(* CoDeSys 2.3.9.28 project: JHV-kovolis.pro *)
(* Libraries: Ethernet.lib 2.12.10 13:48:32, mod_com.lib 2.12.10 13:48:32, ModbusEthernet_04.lib 2.12.10 13:48:36, Standard.lib 2.12.10 13:48:34, SYSLIBCALLBACK.LIB 2.12.10 13:48:32 *)

(* PLC configuration (modules and I/O channels)
IN1 AT %IX0.0 [BOOLOnX_I] Ch_1 Digital input
IN2 AT %IX0.1 [BOOLOnX_I] Ch_2 Digital input
IN3 AT %IX0.2 [BOOLOnX_I] Ch_3 Digital input
IN4 AT %IX0.3 [BOOLOnX_I] Ch_4 Digital input
IN5 AT %IX0.4 [BOOLOnX_I] Ch_5 Digital input
IN6 AT %IX0.5 [BOOLOnX_I] Ch_6 Digital input
IN7 AT %IX0.6 [BOOLOnX_I] Ch_7 Digital input
IN8 AT %IX0.7 [BOOLOnX_I] Ch_8 Digital input
IN9 AT %IX0.8 [BOOLOnX_I] Ch_1 Digital input
IN10 AT %IX0.9 [BOOLOnX_I] Ch_2 Digital input
IN11 AT %IX0.10 [BOOLOnX_I] Ch_3 Digital input
IN12 AT %IX0.11 [BOOLOnX_I] Ch_4 Digital input
IN13 AT %IX0.12 [BOOLOnX_I] Ch_5 Digital input
IN14 AT %IX0.13 [BOOLOnX_I] Ch_6 Digital input
IN15 AT %IX0.14 [BOOLOnX_I] Ch_7 Digital input
IN16 AT %IX0.15 [BOOLOnX_I] Ch_8 Digital input
Fieldbus variables [FB_VARS] node 1, in %IB0 out %QB0
*)

(* Global variable list: Global_Variables *)
VAR_GLOBAL
	IPHost1: STRING:= '192.168.0.100';
	IPHost2: STRING:= '192.168.0.101';

	Host1IN1: BOOL:= FALSE;
	Host1IN2: BOOL:= FALSE;
	Host1IN3: BOOL:= FALSE;
	Host1IN4: BOOL:= FALSE;
	Host1IN5: BOOL:= FALSE;
	Host1IN6: BOOL:= FALSE;
	Host1IN7: BOOL:= FALSE;
	Host1IN8: BOOL:= FALSE;

	Host2IN1: BOOL:= FALSE;
	Host2IN2: BOOL:= FALSE;
	Host2IN3: BOOL:= FALSE;
	Host2IN4: BOOL:= FALSE;
	Host2IN5: BOOL:= FALSE;
	Host2IN6: BOOL:= FALSE;
	Host2IN7: BOOL:= FALSE;
	Host2IN8: BOOL:= FALSE;

	OJS1: ARRAY [1..12] OF STRING;
	OJS2: ARRAY [1..8] OF STRING;
	OJS3: ARRAY [1..16] OF STRING;
	xOJS1: ARRAY [1..12] OF BOOL;
	xOJS2: ARRAY [1..8] OF BOOL;
	xOJS3: ARRAY [1..16] OF BOOL;
	xxOJS1: ARRAY [1..12] OF BOOL; (*Pøevrácená hodnota xOJS1*)
	xxOJS2: ARRAY [1..8] OF BOOL;	(*Pøevrácená hodnota xOJS2*)
	xxOJS3: ARRAY [1..16] OF BOOL;	(*Pøevrácená hodnota xOJS3*)

END_VAR

(* POU PLC_PRG, FBD *)
PROGRAM PLC_PRG
VAR
	Komunikace1: SlaveUDP_IO;
	Komunikace2: SlaveUDP_IO;
	sendStrHost1: ARRAY [1..100] OF WORD;
	sendStrHost2: ARRAY [1..100] OF WORD;
	RecStrHost1: ARRAY [1..100] OF WORD;
	RecStrHost2: ARRAY [1..100] OF WORD;
	Init1: BOOL;
	Init2: BOOL;
	NOERROR1: BOOL;
	NOERROR2: BOOL;
	PrevodnikHost1: WORD_TO_BOOL_16b;
	PrevodnikHost2: WORD_TO_BOOL_16b;
	Slitina: ARRAY [1..2] OF STRING:= 'Slitina1','Slitina2';
END_VAR
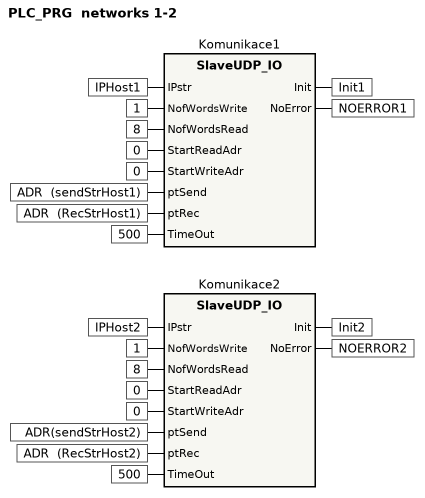
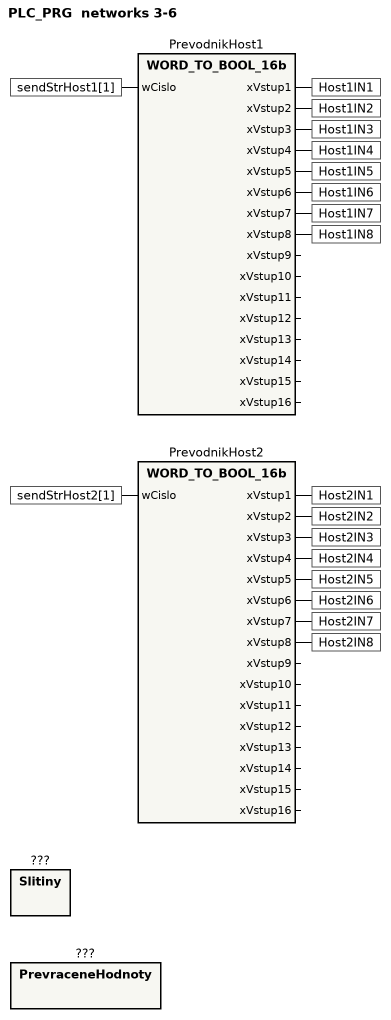
_FBD_ (* Function Block Diagram *)
NETWORK 1
	Komunikace1:SlaveUDP_IO(IPstr: IPHost1, NofWordsWrite: 1, NofWordsRead: 8, StartReadAdr: 0, StartWriteAdr: 0, ptSend: ADR	(sendStrHost1), ptRec: ADR	(RecStrHost1), TimeOut: 500, NoError => NOERROR1) => Init1
NETWORK 2
	Komunikace2:SlaveUDP_IO(IPstr: IPHost2, NofWordsWrite: 1, NofWordsRead: 8, StartReadAdr: 0, StartWriteAdr: 0, ptSend: 	ADR(sendStrHost2), ptRec: ADR	(RecStrHost2), TimeOut: 500, NoError => NOERROR2) => Init2
NETWORK 3
	PrevodnikHost1:WORD_TO_BOOL_16b(wCislo: sendStrHost1[1], xVstup2 => Host1IN2, xVstup3 => Host1IN3, xVstup4 => Host1IN4, xVstup5 => Host1IN5, xVstup6 => Host1IN6, xVstup7 => Host1IN7, xVstup8 => Host1IN8) => Host1IN1
NETWORK 4
	PrevodnikHost2:WORD_TO_BOOL_16b(wCislo: sendStrHost2[1], xVstup2 => Host2IN2, xVstup3 => Host2IN3, xVstup4 => Host2IN4, xVstup5 => Host2IN5, xVstup6 => Host2IN6, xVstup7 => Host2IN7, xVstup8 => Host2IN8) => Host2IN1
NETWORK 5
	???:Slitiny()
NETWORK 6
	???:PrevraceneHodnoty()
_END_FBD_
(* the same logic as Structured Text *)
(* Network 1 *)
Komunikace1(IPstr := IPHost1, NofWordsWrite := 1, NofWordsRead := 8, StartReadAdr := 0, StartWriteAdr := 0, ptSend := ADR	(sendStrHost1), ptRec := ADR	(RecStrHost1), TimeOut := 500);
NOERROR1 := Komunikace1.NoError;
Init1 := Komunikace1.Init;
(* Network 2 *)
Komunikace2(IPstr := IPHost2, NofWordsWrite := 1, NofWordsRead := 8, StartReadAdr := 0, StartWriteAdr := 0, ptSend := 	ADR(sendStrHost2), ptRec := ADR	(RecStrHost2), TimeOut := 500);
NOERROR2 := Komunikace2.NoError;
Init2 := Komunikace2.Init;
(* Network 3 *)
PrevodnikHost1(wCislo := sendStrHost1[1]);
Host1IN2 := PrevodnikHost1.xVstup2;
Host1IN3 := PrevodnikHost1.xVstup3;
Host1IN4 := PrevodnikHost1.xVstup4;
Host1IN5 := PrevodnikHost1.xVstup5;
Host1IN6 := PrevodnikHost1.xVstup6;
Host1IN7 := PrevodnikHost1.xVstup7;
Host1IN8 := PrevodnikHost1.xVstup8;
Host1IN1 := PrevodnikHost1.xVstup1;
(* Network 4 *)
PrevodnikHost2(wCislo := sendStrHost2[1]);
Host2IN2 := PrevodnikHost2.xVstup2;
Host2IN3 := PrevodnikHost2.xVstup3;
Host2IN4 := PrevodnikHost2.xVstup4;
Host2IN5 := PrevodnikHost2.xVstup5;
Host2IN6 := PrevodnikHost2.xVstup6;
Host2IN7 := PrevodnikHost2.xVstup7;
Host2IN8 := PrevodnikHost2.xVstup8;
Host2IN1 := PrevodnikHost2.xVstup1;
(* Network 5: see the listing above *)
(* Network 6: see the listing above *)
END_PROGRAM

(* POU SlaveUDP_IO, ST *)
FUNCTION_BLOCK SlaveUDP_IO
VAR_INPUT
	IPstr:STRING;					(*IP adresa slavu - 750-352,speedwaz etc.*)
	NofWordsWrite:WORD;		(*Pocet wordu, ktere maji byt zapsany*)
	NofWordsRead:WORD;		(*Pocet wordu, tkere maji byt cteny*)
	StartReadAdr:WORD;			(*adresa odkud se bude cist*)
	StartWriteAdr:WORD;			(*odresa kam se bude zapisovat*)
	ptSend:POINTER TO WORD;	(*pointer na pole ktere se bude zapisovat*)
	ptRec:POINTER TO WORD;	(*pointer na pole ktere se bude cist*)
	TimeOut:WORD:=500;		(*cas v milisekundach, pokud neni zadna komunikace, tak potomto case se vystupy nastavi do nuly*)
END_VAR
VAR_OUTPUT
	Init:BOOL;					(*cas do watchdogu byl zapsan a watchdog je spusten -> je mozne komunikovat*)
	NoError:BOOL;			(*zadna chyba pri komunikaci*)
END_VAR
VAR
	state:INT:=0;
	master882: ETHERNET_MODBUSMASTER_UDP;
	start882:BOOL:=FALSE;
	res882:BOOL:=FALSE;
	err882:WORD;
	ready882:BOOL;
	resp882:BYTE;
	ftrig882: F_TRIG;
	tmp_val:WORD;

	ptWrite:POINTER TO BYTE;
	NofWrite:INT;
	WriteAdr:WORD;
END_VAR
IF start882=FALSE THEN
	start882:=TRUE;
	CASE state OF
		0:
			(*zastaveni casovace*)
			tmp_val:=0;
			WriteAdr:=16#100A;
			ptWrite:=ADR(tmp_val);
			NofWrite:=1;
		1:
			(*nastaveni casu, cas je mozne nastavit jen tehdy, kdyz je casovac zastaven*)
			TimeOut:=TimeOut/100;
			tmp_val:=TimeOut;
			NofWordsWrite:=1;
			WriteAdr:=16#1000;
			ptWrite:=ADR(tmp_val);
			NofWrite:=1;
		2:
			(*spusteni watchdogu*)
			tmp_val:=1;
			WriteAdr:=16#100A;
			ptWrite:=ADR(tmp_val);
			NofWrite:=1;
		3:
			(*bezna komunikace*)
			ptWrite:=ptSend;
			NofWrite:=NofWordsWrite;
			WriteAdr:=StartWriteAdr;
	END_CASE;
END_IF;

NofWordsRead;
NofWrite;
IF NofWrite=0 THEN
(*cteni 352 kdyz neni treba nic zapsat*)
master882(strIP_ADDRESS := IPstr,	wPORT := 502,bUNIT_ID := 0,bFUNCTION_CODE := 3,wREAD_ADDRESS := StartReadAdr,wREAD_QUANTITY :=NofWordsRead,
	ptREAD_DATA :=ptRec,wWRITE_ADDRESS := WriteAdr,wWRITE_QUANTITY := NofWrite,ptSEND_DATA :=ptWrite ,xSTART := start882,xRESET := res882,
	tTIME_OUT := t#1s);
ELSE
(*blok pro cteni i zapis v jednom cyklu*)
master882(strIP_ADDRESS := IPstr,	wPORT := 502,bUNIT_ID := 0,bFUNCTION_CODE := 23,wREAD_ADDRESS := StartReadAdr,wREAD_QUANTITY :=NofWordsRead,
	ptREAD_DATA :=ptRec,wWRITE_ADDRESS := WriteAdr,wWRITE_QUANTITY := NofWrite,ptSEND_DATA :=ptWrite ,xSTART := start882,xRESET := res882,
	tTIME_OUT := t#1s);
END_IF;
	(* vystupni promenne *)
	err882:=master882.wERROR;
	ready882:= master882.xREADY;
	resp882:=master882.bRESPONSE_UNIT_ID;

IF master882.wERROR=0 THEN
	NoError:=TRUE;
ELSE
	NoError:=FALSE;
END_IF;
ftrig882(clk:=ready882);
(*prechody ve stavovem automau*)
IF ftrig882.Q   THEN
	 start882:=FALSE;
	IF master882.wERROR=0 THEN
		state:=state+1;	(*neni chyba komunikace, prejdi do dalsiho stavu*)
	ELSE
		IF state>0 AND state<3 THEN
			(*nastala nejaka chyba, vrat so inicializace casovace*)
			state:=0;
		END_IF;
	END_IF;
	IF state>=3 THEN
		state:=3;
		init:=TRUE;
	END_IF;
END_IF;
END_FUNCTION_BLOCK

(* POU Komunikace/WORD_TO_BOOL_16b, ST *)
FUNCTION_BLOCK WORD_TO_BOOL_16b
VAR_INPUT
	wCislo: WORD;

END_VAR
VAR_OUTPUT
	xVstup1: BOOL;
	xVstup2: BOOL;
	xVstup3: BOOL;
	xVstup4: BOOL;
	xVstup5: BOOL;
	xVstup6: BOOL;
	xVstup7: BOOL;
	xVstup8: BOOL;
	xVstup9: BOOL;
	xVstup10: BOOL;
	xVstup11: BOOL;
	xVstup12: BOOL;
	xVstup13: BOOL;
	xVstup14: BOOL;
	xVstup15: BOOL;
	xVstup16: BOOL;
END_VAR
VAR
END_VAR
IF (wCislo > 0)
	THEN
		(*15tı bit*)
		IF(wCislo/32768 > 0)
			THEN
				xVstup16 := TRUE;
				wCislo:= wCislo - 32768;
		ELSE
				xVstup16 := FALSE;
		END_IF

		(*14tı bit*)
		IF(wCislo/16384 > 0)
			THEN
				xVstup15 := TRUE;
				wCislo:= wCislo - 16384;
		ELSE
				xVstup15 := FALSE;
		END_IF

		(*13tı bit*)
		IF(wCislo/8192 > 0)
			THEN
				xVstup14 := TRUE;
				wCislo:= wCislo - 8192;
		ELSE
				xVstup14 := FALSE;
		END_IF

		(*12tı bit*)
		IF(wCislo/4096 > 0)
			THEN
				xVstup13 := TRUE;
				wCislo:= wCislo - 4096;
		ELSE
				xVstup13 := FALSE;
		END_IF

		(*11tı bit*)
		IF(wCislo/2048 > 0)
			THEN
				xVstup12 := TRUE;
				wCislo:= wCislo - 2048;
		ELSE
				xVstup12 := FALSE;
		END_IF

		(*10tı bit*)
		IF(wCislo/1024 > 0)
			THEN
				xVstup11 := TRUE;
				wCislo:= wCislo - 1024;
		ELSE
				xVstup11 := FALSE;
		END_IF

		(*9tı bit*)
		IF(wCislo/512 > 0)
			THEN
				xVstup10 := TRUE;
				wCislo:= wCislo - 512;
		ELSE
				xVstup10 := FALSE;
		END_IF

		(*8tı bit*)
		IF(wCislo/256 > 0)
			THEN
				xVstup9 := TRUE;
				wCislo:= wCislo - 256;
		ELSE
				xVstup9 := FALSE;
		END_IF

		(*7tı bit*)
		IF(wCislo/128 > 0)
			THEN
				xVstup8 := TRUE;
				wCislo:= wCislo - 128;
		ELSE
				xVstup8 := FALSE;
		END_IF

		(*6tı bit*)
		IF(wCislo/64 > 0)
			THEN
				xVstup7 := TRUE;
				wCislo:= wCislo - 64;
		ELSE
				xVstup7 := FALSE;
		END_IF

		(*5tı bit*)
		IF(wCislo/32 > 0)
			THEN
				xVstup6 := TRUE;
				wCislo:= wCislo - 32;
		ELSE
				xVstup6 := FALSE;
		END_IF

		(*4tı bit*)
		IF(wCislo/16 > 0)
			THEN
				xVstup5 := TRUE;
				wCislo:= wCislo - 16;
		ELSE
				xVstup5 := FALSE;
		END_IF

		(*3tí bit*)
		IF(wCislo/8 > 0)
			THEN
				xVstup4 := TRUE;
				wCislo:= wCislo - 8;
		ELSE
				xVstup4 := FALSE;
		END_IF

		(*2hı bit*)
		IF(wCislo/4 > 0)
			THEN
				xVstup3 := TRUE;
				wCislo:= wCislo - 4;
		ELSE
				xVstup3 := FALSE;
		END_IF

		(*1ní bit*)
		IF(wCislo/2 > 0)
			THEN
				xVstup2 := TRUE;
				wCislo:= wCislo - 2;
		ELSE
				xVstup2 := FALSE;
		END_IF

		(*0tı bit*)
		IF(wCislo > 0)
			THEN
				xVstup1 := TRUE;
				wCislo:= wCislo - 1;
		ELSE
				xVstup1 := FALSE;
		END_IF
END_IF
END_FUNCTION_BLOCK

(* POU Slitiny/Slitiny, CFC *)
PROGRAM Slitiny
VAR
	s1: VybranaSlitina;
	s2: VybranaSlitina;
	s3: VybranaSlitina;
	s4: VybranaSlitina;
	s5: VybranaSlitina;
	s6: VybranaSlitina;
	s7: VybranaSlitina;
	s8: VybranaSlitina;
	s9: VybranaSlitina;
	s10: VybranaSlitina;
	s11: VybranaSlitina;
	s12: VybranaSlitina;

	s13: VybranaSlitina;
	s14: VybranaSlitina;
	s15: VybranaSlitina;
	s16: VybranaSlitina;
	s17: VybranaSlitina;
	s18: VybranaSlitina;
	s19: VybranaSlitina;
	s20: VybranaSlitina;

	s21: VybranaSlitina;
	s22: VybranaSlitina;
	s23: VybranaSlitina;
	s24: VybranaSlitina;
	s25: VybranaSlitina;
	s26: VybranaSlitina;
	s27: VybranaSlitina;
	s28: VybranaSlitina;
	s29: VybranaSlitina;
	s30: VybranaSlitina;
	s31: VybranaSlitina;
	s32: VybranaSlitina;
	s33: VybranaSlitina;
	s34: VybranaSlitina;
	s35: VybranaSlitina;
END_VAR
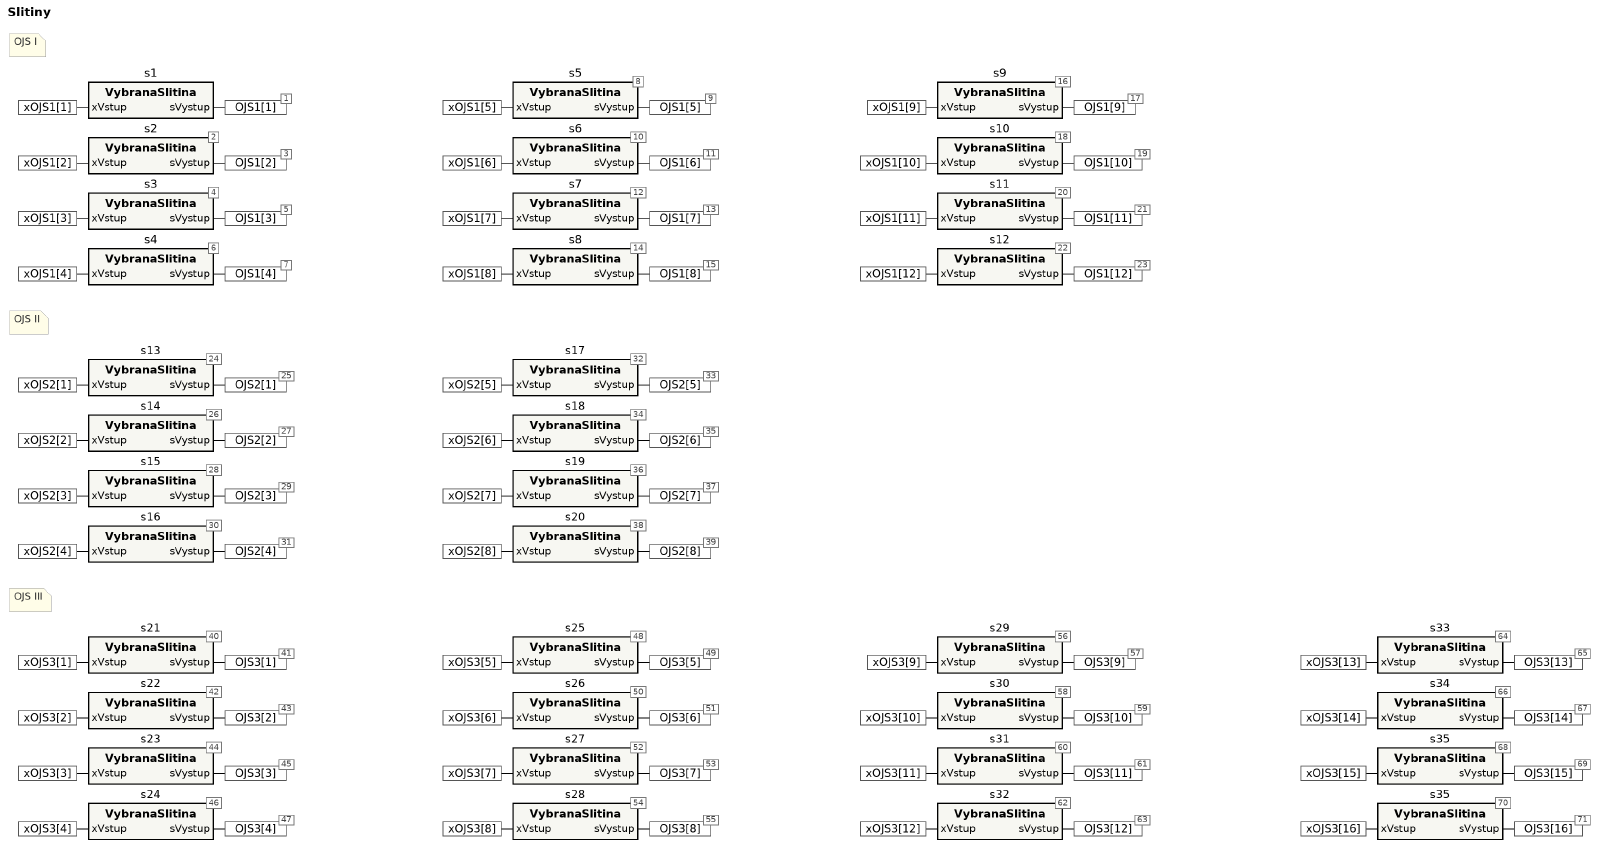
_CFC_ (* Continuous Function Chart, elements in execution order *)
(* OJS I *)
#0 s1:VybranaSlitina(xVstup: xOJS1[1])
#1 OJS1[1] <= #0.sVystup
#2 s2:VybranaSlitina(xVstup: xOJS1[2])
#3 OJS1[2] <= #2.sVystup
#4 s3:VybranaSlitina(xVstup: xOJS1[3])
#5 OJS1[3] <= #4.sVystup
#6 s4:VybranaSlitina(xVstup: xOJS1[4])
#7 OJS1[4] <= #6.sVystup
#8 s5:VybranaSlitina(xVstup: xOJS1[5])
#9 OJS1[5] <= #8.sVystup
#10 s6:VybranaSlitina(xVstup: xOJS1[6])
#11 OJS1[6] <= #10.sVystup
#12 s7:VybranaSlitina(xVstup: xOJS1[7])
#13 OJS1[7] <= #12.sVystup
#14 s8:VybranaSlitina(xVstup: xOJS1[8])
#15 OJS1[8] <= #14.sVystup
#16 s9:VybranaSlitina(xVstup: xOJS1[9])
#17 OJS1[9] <= #16.sVystup
#18 s10:VybranaSlitina(xVstup: xOJS1[10])
#19 OJS1[10] <= #18.sVystup
#20 s11:VybranaSlitina(xVstup: xOJS1[11])
#21 OJS1[11] <= #20.sVystup
#22 s12:VybranaSlitina(xVstup: xOJS1[12])
#23 OJS1[12] <= #22.sVystup
(* OJS II *)
#24 s13:VybranaSlitina(xVstup: xOJS2[1])
#25 OJS2[1] <= #24.sVystup
#26 s14:VybranaSlitina(xVstup: xOJS2[2])
#27 OJS2[2] <= #26.sVystup
#28 s15:VybranaSlitina(xVstup: xOJS2[3])
#29 OJS2[3] <= #28.sVystup
#30 s16:VybranaSlitina(xVstup: xOJS2[4])
#31 OJS2[4] <= #30.sVystup
#32 s17:VybranaSlitina(xVstup: xOJS2[5])
#33 OJS2[5] <= #32.sVystup
#34 s18:VybranaSlitina(xVstup: xOJS2[6])
#35 OJS2[6] <= #34.sVystup
#36 s19:VybranaSlitina(xVstup: xOJS2[7])
#37 OJS2[7] <= #36.sVystup
#38 s20:VybranaSlitina(xVstup: xOJS2[8])
#39 OJS2[8] <= #38.sVystup
(* OJS III *)
#40 s21:VybranaSlitina(xVstup: xOJS3[1])
#41 OJS3[1] <= #40.sVystup
#42 s22:VybranaSlitina(xVstup: xOJS3[2])
#43 OJS3[2] <= #42.sVystup
#44 s23:VybranaSlitina(xVstup: xOJS3[3])
#45 OJS3[3] <= #44.sVystup
#46 s24:VybranaSlitina(xVstup: xOJS3[4])
#47 OJS3[4] <= #46.sVystup
#48 s25:VybranaSlitina(xVstup: xOJS3[5])
#49 OJS3[5] <= #48.sVystup
#50 s26:VybranaSlitina(xVstup: xOJS3[6])
#51 OJS3[6] <= #50.sVystup
#52 s27:VybranaSlitina(xVstup: xOJS3[7])
#53 OJS3[7] <= #52.sVystup
#54 s28:VybranaSlitina(xVstup: xOJS3[8])
#55 OJS3[8] <= #54.sVystup
#56 s29:VybranaSlitina(xVstup: xOJS3[9])
#57 OJS3[9] <= #56.sVystup
#58 s30:VybranaSlitina(xVstup: xOJS3[10])
#59 OJS3[10] <= #58.sVystup
#60 s31:VybranaSlitina(xVstup: xOJS3[11])
#61 OJS3[11] <= #60.sVystup
#62 s32:VybranaSlitina(xVstup: xOJS3[12])
#63 OJS3[12] <= #62.sVystup
#64 s33:VybranaSlitina(xVstup: xOJS3[13])
#65 OJS3[13] <= #64.sVystup
#66 s34:VybranaSlitina(xVstup: xOJS3[14])
#67 OJS3[14] <= #66.sVystup
#68 s35:VybranaSlitina(xVstup: xOJS3[15])
#69 OJS3[15] <= #68.sVystup
#70 s35:VybranaSlitina(xVstup: xOJS3[16])
#71 OJS3[16] <= #70.sVystup
_END_CFC_
END_PROGRAM

(* POU Slitiny/VybranaSlitina, ST *)
FUNCTION_BLOCK VybranaSlitina
VAR_INPUT
	xVstup: BOOL;
END_VAR
VAR_OUTPUT
	sVystup: STRING;
END_VAR
VAR
END_VAR
IF (xVstup)
THEN
	sVystup:= PLC_PRG.Slitina[1];
ELSE
	sVystup:= PLC_PRG.Slitina[2];
END_IF
END_FUNCTION_BLOCK

(* POU Slitiny/PrevraceneHodnoty, CFC *)
PROGRAM PrevraceneHodnoty
VAR
END_VAR
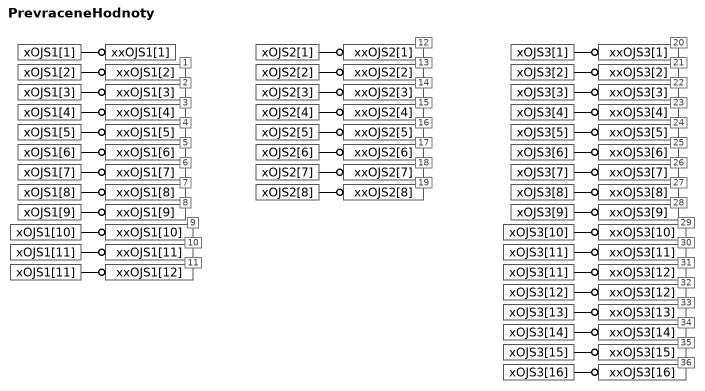
_CFC_ (* Continuous Function Chart, elements in execution order *)
#0 xxOJS1[1] <= NOT xOJS1[1]
#1 xxOJS1[2] <= NOT xOJS1[2]
#2 xxOJS1[3] <= NOT xOJS1[3]
#3 xxOJS1[4] <= NOT xOJS1[4]
#4 xxOJS1[5] <= NOT xOJS1[5]
#5 xxOJS1[6] <= NOT xOJS1[6]
#6 xxOJS1[7] <= NOT xOJS1[7]
#7 xxOJS1[8] <= NOT xOJS1[8]
#8 xxOJS1[9] <= NOT xOJS1[9]
#9 xxOJS1[10] <= NOT xOJS1[10]
#10 xxOJS1[11] <= NOT xOJS1[11]
#11 xxOJS1[12] <= NOT xOJS1[11]
#12 xxOJS2[1] <= NOT xOJS2[1]
#13 xxOJS2[2] <= NOT xOJS2[2]
#14 xxOJS2[3] <= NOT xOJS2[3]
#15 xxOJS2[4] <= NOT xOJS2[4]
#16 xxOJS2[5] <= NOT xOJS2[5]
#17 xxOJS2[6] <= NOT xOJS2[6]
#18 xxOJS2[7] <= NOT xOJS2[7]
#19 xxOJS2[8] <= NOT xOJS2[8]
#20 xxOJS3[1] <= NOT xOJS3[1]
#21 xxOJS3[2] <= NOT xOJS3[2]
#22 xxOJS3[3] <= NOT xOJS3[3]
#23 xxOJS3[4] <= NOT xOJS3[4]
#24 xxOJS3[5] <= NOT xOJS3[5]
#25 xxOJS3[6] <= NOT xOJS3[6]
#26 xxOJS3[7] <= NOT xOJS3[7]
#27 xxOJS3[8] <= NOT xOJS3[8]
#28 xxOJS3[9] <= NOT xOJS3[9]
#29 xxOJS3[10] <= NOT xOJS3[10]
#30 xxOJS3[11] <= NOT xOJS3[11]
#31 xxOJS3[12] <= NOT xOJS3[11]
#32 xxOJS3[12] <= NOT xOJS3[12]
#33 xxOJS3[13] <= NOT xOJS3[13]
#34 xxOJS3[14] <= NOT xOJS3[14]
#35 xxOJS3[15] <= NOT xOJS3[15]
#36 xxOJS3[16] <= NOT xOJS3[16]
_END_CFC_
(* the same logic as Structured Text *)
xxOJS1[1] := NOT xOJS1[1];
xxOJS1[2] := NOT xOJS1[2];
xxOJS1[3] := NOT xOJS1[3];
xxOJS1[4] := NOT xOJS1[4];
xxOJS1[5] := NOT xOJS1[5];
xxOJS1[6] := NOT xOJS1[6];
xxOJS1[7] := NOT xOJS1[7];
xxOJS1[8] := NOT xOJS1[8];
xxOJS1[9] := NOT xOJS1[9];
xxOJS1[10] := NOT xOJS1[10];
xxOJS1[11] := NOT xOJS1[11];
xxOJS1[12] := NOT xOJS1[11];
xxOJS2[1] := NOT xOJS2[1];
xxOJS2[2] := NOT xOJS2[2];
xxOJS2[3] := NOT xOJS2[3];
xxOJS2[4] := NOT xOJS2[4];
xxOJS2[5] := NOT xOJS2[5];
xxOJS2[6] := NOT xOJS2[6];
xxOJS2[7] := NOT xOJS2[7];
xxOJS2[8] := NOT xOJS2[8];
xxOJS3[1] := NOT xOJS3[1];
xxOJS3[2] := NOT xOJS3[2];
xxOJS3[3] := NOT xOJS3[3];
xxOJS3[4] := NOT xOJS3[4];
xxOJS3[5] := NOT xOJS3[5];
xxOJS3[6] := NOT xOJS3[6];
xxOJS3[7] := NOT xOJS3[7];
xxOJS3[8] := NOT xOJS3[8];
xxOJS3[9] := NOT xOJS3[9];
xxOJS3[10] := NOT xOJS3[10];
xxOJS3[11] := NOT xOJS3[11];
xxOJS3[12] := NOT xOJS3[11];
xxOJS3[12] := NOT xOJS3[12];
xxOJS3[13] := NOT xOJS3[13];
xxOJS3[14] := NOT xOJS3[14];
xxOJS3[15] := NOT xOJS3[15];
xxOJS3[16] := NOT xOJS3[16];
END_PROGRAM

(* POU Komunikace/BOOL_TO_WORD_16b, CFC *)
FUNCTION_BLOCK BOOL_TO_WORD_16b
VAR_INPUT
	xVystup1: BOOL;
	xVystup2: BOOL;
	xVystup3: BOOL;
	xVystup4: BOOL;
	xVystup5: BOOL;
	xVystup6: BOOL;
	xVystup7: BOOL;
	xVystup8: BOOL;
	xVystup9: BOOL;
	xVystup10: BOOL;
	xVystup11: BOOL;
	xVystup12: BOOL;
	xVystup13: BOOL;
	xVystup14: BOOL;
	xVystup15: BOOL;
	xVystup16: BOOL;
END_VAR
VAR
END_VAR
VAR_OUTPUT
	wVystup: WORD;
END_VAR
VAR (* helpers for the ST form of the networks *)
	_t1 : WORD;
	_t8 : WORD;
	_t11 : WORD;
	_t14 : WORD;
	_t18 : WORD;
	_t21 : WORD;
	_t24 : WORD;
	_t27 : WORD;
	_t30 : WORD;
	_t33 : WORD;
	_t36 : WORD;
	_t39 : WORD;
	_t42 : WORD;
	_t45 : WORD;
	_t48 : WORD;
	_t6 : WORD;
END_VAR
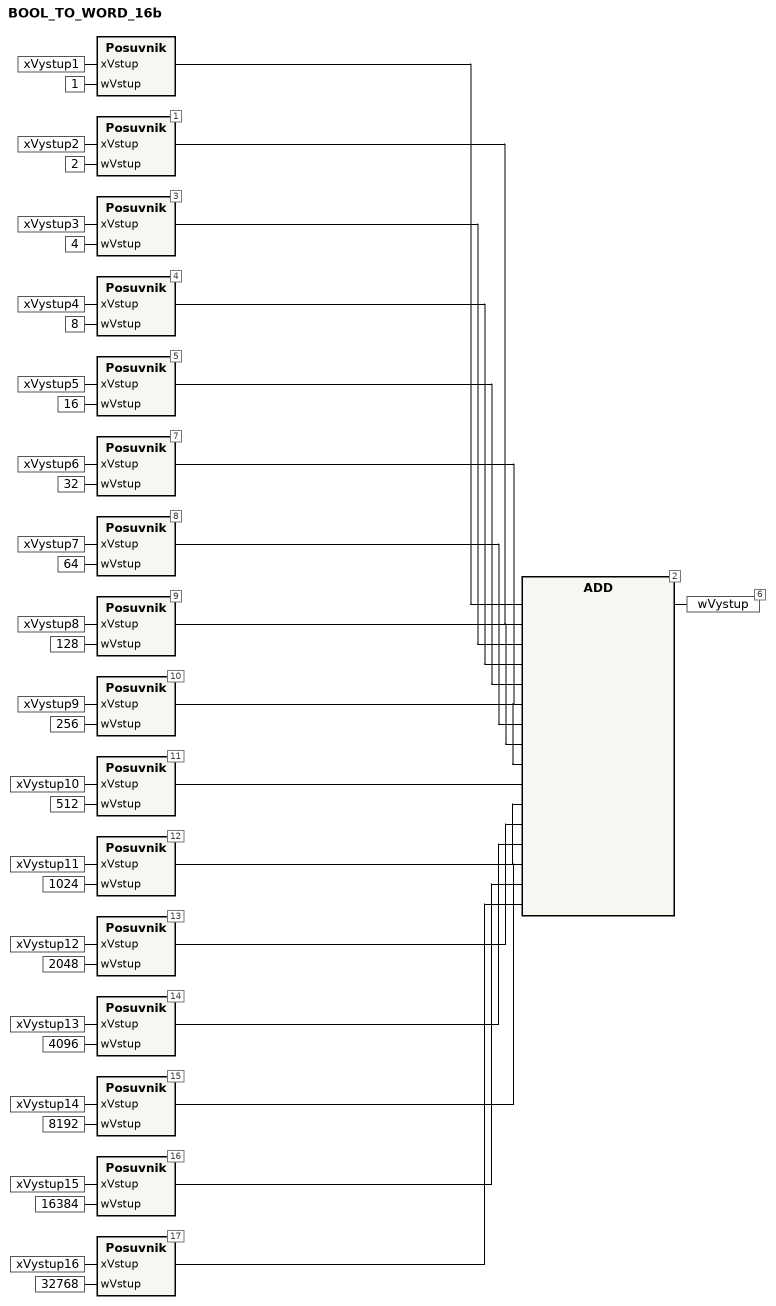
_CFC_ (* Continuous Function Chart, elements in execution order *)
#0 Posuvnik(xVstup: xVystup1, wVstup: 1)
#1 Posuvnik(xVstup: xVystup2, wVstup: 2)
#2 ADD(#0, #1, #3, #4, #5, #7, #8, #9, #10, #11, #12, #13, #14, #15, #16, #17)
#3 Posuvnik(xVstup: xVystup3, wVstup: 4)
#4 Posuvnik(xVstup: xVystup4, wVstup: 8)
#5 Posuvnik(xVstup: xVystup5, wVstup: 16)
#6 wVystup <= #2
#7 Posuvnik(xVstup: xVystup6, wVstup: 32)
#8 Posuvnik(xVstup: xVystup7, wVstup: 64)
#9 Posuvnik(xVstup: xVystup8, wVstup: 128)
#10 Posuvnik(xVstup: xVystup9, wVstup: 256)
#11 Posuvnik(xVstup: xVystup10, wVstup: 512)
#12 Posuvnik(xVstup: xVystup11, wVstup: 1024)
#13 Posuvnik(xVstup: xVystup12, wVstup: 2048)
#14 Posuvnik(xVstup: xVystup13, wVstup: 4096)
#15 Posuvnik(xVstup: xVystup14, wVstup: 8192)
#16 Posuvnik(xVstup: xVystup15, wVstup: 16384)
#17 Posuvnik(xVstup: xVystup16, wVstup: 32768)
_END_CFC_
(* the same logic as Structured Text *)
_t1 := Posuvnik(xVstup := xVystup1, wVstup := 1);
_t6 := _t1 + Posuvnik(xVstup := xVystup2, wVstup := 2) + _t8 + _t11 + _t14 + _t18 + _t21 + _t24 + _t27 + _t30 + _t33 + _t36 + _t39 + _t42 + _t45 + _t48;
_t8 := Posuvnik(xVstup := xVystup3, wVstup := 4);
_t11 := Posuvnik(xVstup := xVystup4, wVstup := 8);
_t14 := Posuvnik(xVstup := xVystup5, wVstup := 16);
wVystup := _t6;
_t18 := Posuvnik(xVstup := xVystup6, wVstup := 32);
_t21 := Posuvnik(xVstup := xVystup7, wVstup := 64);
_t24 := Posuvnik(xVstup := xVystup8, wVstup := 128);
_t27 := Posuvnik(xVstup := xVystup9, wVstup := 256);
_t30 := Posuvnik(xVstup := xVystup10, wVstup := 512);
_t33 := Posuvnik(xVstup := xVystup11, wVstup := 1024);
_t36 := Posuvnik(xVstup := xVystup12, wVstup := 2048);
_t39 := Posuvnik(xVstup := xVystup13, wVstup := 4096);
_t42 := Posuvnik(xVstup := xVystup14, wVstup := 8192);
_t45 := Posuvnik(xVstup := xVystup15, wVstup := 16384);
_t48 := Posuvnik(xVstup := xVystup16, wVstup := 32768);
END_FUNCTION_BLOCK

(* POU Komunikace/Posuvnik, ST *)
FUNCTION Posuvnik : WORD
VAR_INPUT
	xVstup: BOOL;
	wVstup: WORD;
END_VAR
VAR
END_VAR
IF (xVstup = TRUE)
THEN
Posuvnik := wVstup;
ELSE
Posuvnik := 0;
END_IF
END_FUNCTION

(* Visualisation Nastaveni
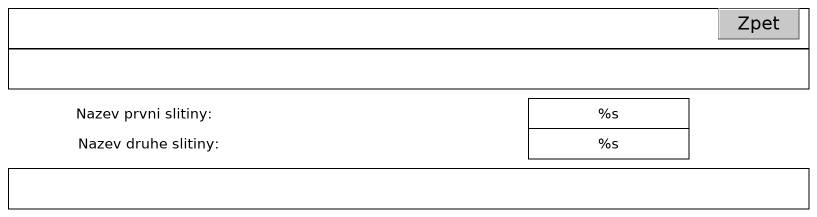
rectangle at (0,0)-(801,41): text "NASTAVENI"
button at (710,0)-(791,31): text "Zpet"; opens plc_vizu
rectangle at (0,40)-(801,81): text "Slitiny:"
rectangle at (30,90)-(251,121): text "Nazev prvni slitiny:"
rectangle at (30,120)-(251,151): text "Nazev druhe slitiny:"
rectangle at (520,90)-(681,121): text "%s"; shows PLC_PRG.Slitina[1]; editable
rectangle at (520,120)-(681,151): text "%s"; shows PLC_PRG.Slitina[2]; editable
rectangle at (0,160)-(801,201): text "Slitiny:"
*)

(* Visualisation OJS1/OJS_I
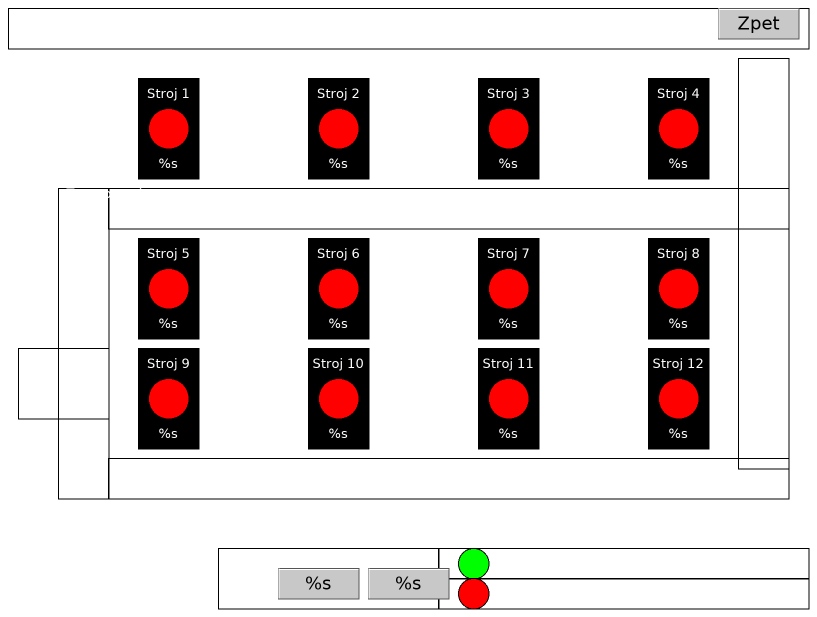
rectangle at (60,170)-(171,201): text "Transportní cesta"
rectangle at (130,70)-(191,101): text "Stroj 1"
ellipse at (140,100)-(181,141): alarm colour if IN1
rectangle at (640,70)-(701,101): text "Stroj 4"
rectangle at (300,70)-(361,101): text "Stroj 2"
rectangle at (470,70)-(531,101): text "Stroj 3"
rectangle at (130,230)-(191,261): text "Stroj 5"
rectangle at (300,230)-(361,261): text "Stroj 6"
rectangle at (470,230)-(531,261): text "Stroj 7"
rectangle at (640,230)-(701,261): text "Stroj 8"
rectangle at (130,340)-(191,371): text "Stroj 9"
rectangle at (300,340)-(361,371): text "Stroj 10"
rectangle at (470,340)-(531,371): text "Stroj 11"
rectangle at (640,340)-(701,371): text "Stroj 12"
rectangle at (0,0)-(801,41): text "SLEVARNA AL OJS I"
button at (710,0)-(791,31): text "Zpet"; opens plc_vizu
rectangle at (300,140)-(361,171): text "%s"; shows OJS1[2]; toggles xOJS1[2]
rectangle at (130,140)-(191,171): text "%s"; shows OJS1[1]; toggles xOJS1[1]
rectangle at (640,140)-(701,171): text "%s"; shows OJS1[4]; toggles xOJS1[4]
rectangle at (130,300)-(191,331): text "%s"; shows OJS1[5]; toggles xOJS1[5]
rectangle at (300,300)-(361,331): text "%s"; shows OJS1[6]; toggles xOJS1[6]
rectangle at (470,300)-(531,331): text "%s"; shows OJS1[7]; toggles xOJS1[7]
rectangle at (640,300)-(701,331): text "%s"; shows OJS1[8]; toggles xOJS1[8]
rectangle at (130,410)-(191,441): text "%s"; shows OJS1[9]; toggles xOJS1[9]
rectangle at (300,410)-(361,441): text "%s"; shows OJS1[10]; toggles xOJS1[10]
rectangle at (470,410)-(531,441): text "%s"; shows OJS1[11]; toggles xOJS1[11]
rectangle at (640,410)-(701,441): text "%s"; shows OJS1[12]; toggles xOJS1[12]
ellipse at (310,100)-(351,141): alarm colour if IN2
ellipse at (480,100)-(521,141): alarm colour if IN3
ellipse at (650,100)-(691,141): alarm colour if IN4
ellipse at (140,260)-(181,301): alarm colour if IN5
ellipse at (310,260)-(351,301): alarm colour if IN6
ellipse at (480,260)-(521,301): alarm colour if IN7
ellipse at (650,260)-(691,301): alarm colour if IN8
ellipse at (140,370)-(181,411): alarm colour if IN9
ellipse at (310,370)-(351,411): alarm colour if IN10
ellipse at (480,370)-(521,411): alarm colour if IN11
ellipse at (650,370)-(691,411): alarm colour if IN12
rectangle at (430,540)-(801,571): text "Stroj má dostatatek materialu na vyrobu"
rectangle at (430,570)-(801,601): text "Stroj ocekava slitinu hliniku"
rectangle at (210,540)-(431,601): text "Filtrovat:"
button at (360,560)-(441,591): text "%s"; shows PLC_PRG.Slitina[2]; opens OJS_I_FS2
button at (270,560)-(351,591): text "%s"; shows PLC_PRG.Slitina[1]; opens OJS_I_FS1
rectangle at (470,140)-(531,171): text "%s"; shows OJS1[3]; toggles xOJS1[3]
21 more shapes without text or variables
*)

(* Visualisation OJS1/OJS_I_FS1
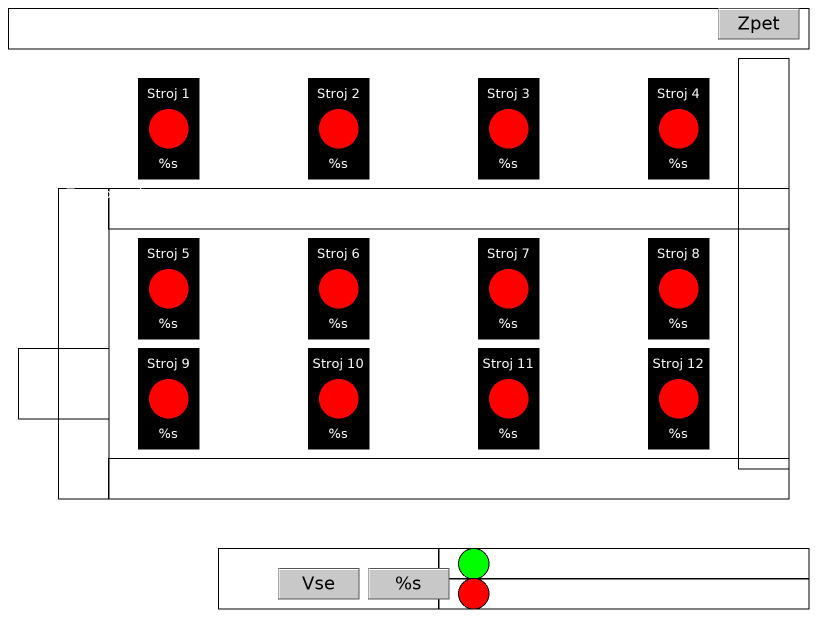
rectangle at (60,170)-(171,201): text "Transportní cesta"
rectangle at (130,70)-(191,101): text "Stroj 1"
ellipse at (140,100)-(181,141): alarm colour if IN1
rectangle at (640,70)-(701,101): text "Stroj 4"
rectangle at (300,70)-(361,101): text "Stroj 2"
rectangle at (470,70)-(531,101): text "Stroj 3"
rectangle at (130,230)-(191,261): text "Stroj 5"
rectangle at (300,230)-(361,261): text "Stroj 6"
rectangle at (470,230)-(531,261): text "Stroj 7"
rectangle at (640,230)-(701,261): text "Stroj 8"
rectangle at (130,340)-(191,371): text "Stroj 9"
rectangle at (300,340)-(361,371): text "Stroj 10"
rectangle at (470,340)-(531,371): text "Stroj 11"
rectangle at (640,340)-(701,371): text "Stroj 12"
rectangle at (0,0)-(801,41): text "SLEVARNA AL OJS I - FILTR"
button at (710,0)-(791,31): text "Zpet"; opens plc_vizu
rectangle at (130,140)-(191,171): text "%s"; shows OJS1[1]; toggles xOJS1[1]
rectangle at (300,140)-(361,171): text "%s"; shows OJS1[2]; toggles xOJS1[2]
rectangle at (470,140)-(531,171): text "%s"; shows OJS1[3]; toggles xOJS1[3]
rectangle at (640,140)-(701,171): text "%s"; shows OJS1[4]; toggles xOJS1[4]
rectangle at (130,300)-(191,331): text "%s"; shows OJS1[5]; toggles xOJS1[5]
rectangle at (300,300)-(361,331): text "%s"; shows OJS1[6]; toggles xOJS1[6]
rectangle at (470,300)-(531,331): text "%s"; shows OJS1[7]; toggles xOJS1[7]
rectangle at (640,300)-(701,331): text "%s"; shows OJS1[8]; toggles xOJS1[8]
rectangle at (130,410)-(191,441): text "%s"; shows OJS1[9]; toggles xOJS1[9]
rectangle at (300,410)-(361,441): text "%s"; shows OJS1[10]; toggles xOJS1[10]
rectangle at (470,410)-(531,441): text "%s"; shows OJS1[11]; toggles xOJS1[11]
rectangle at (640,410)-(701,441): text "%s"; shows OJS1[12]; toggles xOJS1[12]
ellipse at (310,100)-(351,141): alarm colour if IN2
ellipse at (480,100)-(521,141): alarm colour if IN3
ellipse at (650,100)-(691,141): alarm colour if IN4
ellipse at (140,260)-(181,301): alarm colour if IN5
ellipse at (310,260)-(351,301): alarm colour if IN6
ellipse at (480,260)-(521,301): alarm colour if IN7
ellipse at (650,260)-(691,301): alarm colour if IN8
ellipse at (140,370)-(181,411): alarm colour if IN9
ellipse at (310,370)-(351,411): alarm colour if IN10
ellipse at (480,370)-(521,411): alarm colour if IN11
ellipse at (650,370)-(691,411): alarm colour if IN12
rectangle at (430,540)-(801,571): text "Stroj má dostatatek materialu na vyrobu"
rectangle at (430,570)-(801,601): text "Stroj ocekava slitinu hliniku"
rectangle at (210,540)-(431,601): text "Filtrovat:"
button at (360,560)-(441,591): text "%s"; shows PLC_PRG.Slitina[2]; opens OJS_I_FS2
button at (270,560)-(351,591): text "Vse"; opens OJS_I
rectangle at (350,0)-(511,41): text "%s"; shows PLC_PRG.Slitina[1]
rectangle at (130,60)-(191,181): alarm colour if xxOJS1[1]
rectangle at (300,60)-(361,181): alarm colour if xxOJS1[2]
rectangle at (470,60)-(531,181): alarm colour if xxOJS1[3]
rectangle at (640,60)-(701,181): alarm colour if xxOJS1[4]
rectangle at (130,220)-(191,341): alarm colour if xxOJS1[5]
rectangle at (300,220)-(361,341): alarm colour if xxOJS1[6]
rectangle at (470,220)-(531,341): alarm colour if xxOJS1[7]
rectangle at (640,220)-(701,341): alarm colour if xxOJS1[8]
rectangle at (130,330)-(191,451): alarm colour if xxOJS1[9]
rectangle at (300,330)-(361,451): alarm colour if xxOJS1[10]
rectangle at (470,330)-(531,451): alarm colour if xxOJS1[11]
rectangle at (640,330)-(701,451): alarm colour if xxOJS1[12]
21 more shapes without text or variables
*)

(* Visualisation OJS1/OJS_I_FS1x
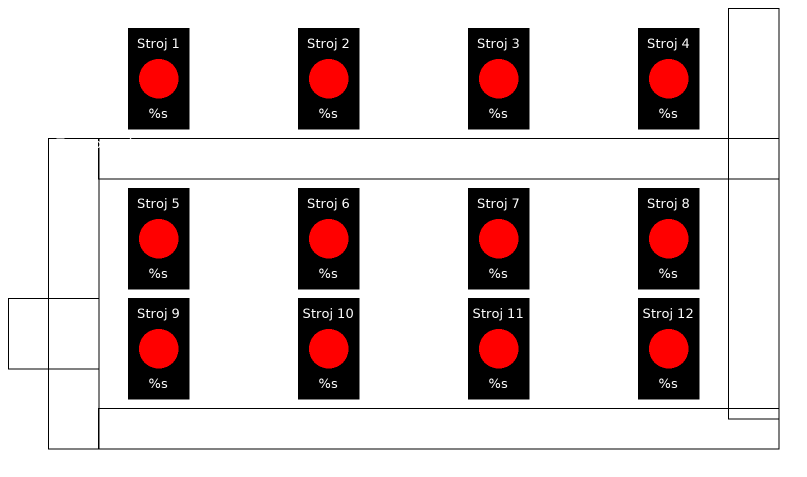
rectangle at (50,120)-(161,151): text "Transportní cesta"
rectangle at (120,20)-(181,51): text "Stroj 1"
ellipse at (130,50)-(171,91): alarm colour if IN1
rectangle at (630,20)-(691,51): text "Stroj 4"
rectangle at (290,20)-(351,51): text "Stroj 2"
rectangle at (460,20)-(521,51): text "Stroj 3"
rectangle at (120,180)-(181,211): text "Stroj 5"
rectangle at (290,180)-(351,211): text "Stroj 6"
rectangle at (460,180)-(521,211): text "Stroj 7"
rectangle at (630,180)-(691,211): text "Stroj 8"
rectangle at (120,290)-(181,321): text "Stroj 9"
rectangle at (290,290)-(351,321): text "Stroj 10"
rectangle at (460,290)-(521,321): text "Stroj 11"
rectangle at (630,290)-(691,321): text "Stroj 12"
rectangle at (120,90)-(181,121): text "%s"; shows OJS1[1]; toggles xOJS1[1]
rectangle at (290,90)-(351,121): text "%s"; shows OJS1[2]; toggles xOJS1[2]
rectangle at (460,90)-(521,121): text "%s"; shows OJS1[3]; toggles xOJS1[3]
rectangle at (630,90)-(691,121): text "%s"; shows OJS1[4]; toggles xOJS1[4]
rectangle at (120,250)-(181,281): text "%s"; shows OJS1[5]; toggles xOJS1[5]
rectangle at (290,250)-(351,281): text "%s"; shows OJS1[6]; toggles xOJS1[6]
rectangle at (460,250)-(521,281): text "%s"; shows OJS1[7]; toggles xOJS1[7]
rectangle at (630,250)-(691,281): text "%s"; shows OJS1[8]; toggles xOJS1[8]
rectangle at (120,360)-(181,391): text "%s"; shows OJS1[9]; toggles xOJS1[9]
rectangle at (290,360)-(351,391): text "%s"; shows OJS1[10]; toggles xOJS1[10]
rectangle at (460,360)-(521,391): text "%s"; shows OJS1[11]; toggles xOJS1[11]
rectangle at (630,360)-(691,391): text "%s"; shows OJS1[12]; toggles xOJS1[12]
ellipse at (300,50)-(341,91): alarm colour if IN2
ellipse at (470,50)-(511,91): alarm colour if IN3
ellipse at (640,50)-(681,91): alarm colour if IN4
ellipse at (130,210)-(171,251): alarm colour if IN5
ellipse at (300,210)-(341,251): alarm colour if IN6
ellipse at (470,210)-(511,251): alarm colour if IN7
ellipse at (640,210)-(681,251): alarm colour if IN8
ellipse at (130,320)-(171,361): alarm colour if IN9
ellipse at (300,320)-(341,361): alarm colour if IN10
ellipse at (470,320)-(511,361): alarm colour if IN11
ellipse at (640,320)-(681,361): alarm colour if IN12
rectangle at (120,10)-(181,131): alarm colour if xxOJS1[1]
rectangle at (290,10)-(351,131): alarm colour if xxOJS1[2]
rectangle at (460,10)-(521,131): alarm colour if xxOJS1[3]
rectangle at (630,10)-(691,131): alarm colour if xxOJS1[4]
rectangle at (120,170)-(181,291): alarm colour if xxOJS1[5]
rectangle at (290,170)-(351,291): alarm colour if xxOJS1[6]
rectangle at (460,170)-(521,291): alarm colour if xxOJS1[7]
rectangle at (630,170)-(691,291): alarm colour if xxOJS1[8]
rectangle at (120,280)-(181,401): alarm colour if xxOJS1[9]
rectangle at (290,280)-(351,401): alarm colour if xxOJS1[10]
rectangle at (460,280)-(521,401): alarm colour if xxOJS1[11]
rectangle at (630,280)-(691,401): alarm colour if xxOJS1[12]
19 more shapes without text or variables
*)

(* Visualisation OJS1/OJS_I_FS2
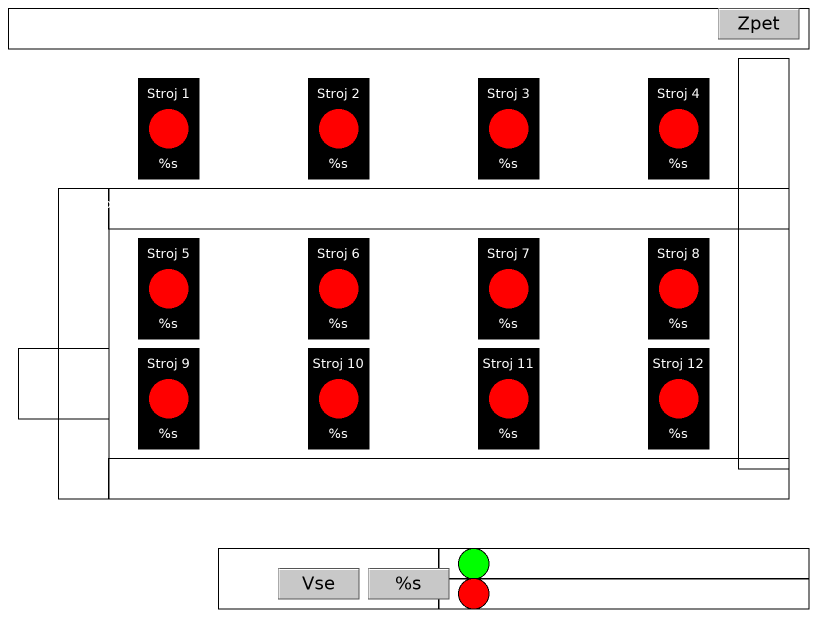
rectangle at (60,180)-(171,211): text "Transportní cesta"
rectangle at (130,70)-(191,101): text "Stroj 1"
ellipse at (140,100)-(181,141): alarm colour if IN1
rectangle at (640,70)-(701,101): text "Stroj 4"
rectangle at (300,70)-(361,101): text "Stroj 2"
rectangle at (470,70)-(531,101): text "Stroj 3"
rectangle at (130,230)-(191,261): text "Stroj 5"
rectangle at (300,230)-(361,261): text "Stroj 6"
rectangle at (470,230)-(531,261): text "Stroj 7"
rectangle at (640,230)-(701,261): text "Stroj 8"
rectangle at (130,340)-(191,371): text "Stroj 9"
rectangle at (300,340)-(361,371): text "Stroj 10"
rectangle at (470,340)-(531,371): text "Stroj 11"
rectangle at (640,340)-(701,371): text "Stroj 12"
rectangle at (0,0)-(801,41): text "SLEVARNA AL OJS I - FILTR"
button at (710,0)-(791,31): text "Zpet"; opens plc_vizu
rectangle at (130,140)-(191,171): text "%s"; shows OJS1[1]; toggles xOJS1[1]
rectangle at (300,140)-(361,171): text "%s"; shows OJS1[2]; toggles xOJS1[2]
rectangle at (470,140)-(531,171): text "%s"; shows OJS1[3]; toggles xOJS1[3]
rectangle at (640,140)-(701,171): text "%s"; shows OJS1[4]; toggles xOJS1[4]
rectangle at (130,300)-(191,331): text "%s"; shows OJS1[5]; toggles xOJS1[5]
rectangle at (300,300)-(361,331): text "%s"; shows OJS1[6]; toggles xOJS1[6]
rectangle at (470,300)-(531,331): text "%s"; shows OJS1[7]; toggles xOJS1[7]
rectangle at (640,300)-(701,331): text "%s"; shows OJS1[8]; toggles xOJS1[8]
rectangle at (130,410)-(191,441): text "%s"; shows OJS1[9]; toggles xOJS1[9]
rectangle at (300,410)-(361,441): text "%s"; shows OJS1[10]; toggles xOJS1[10]
rectangle at (470,410)-(531,441): text "%s"; shows OJS1[11]; toggles xOJS1[11]
rectangle at (640,410)-(701,441): text "%s"; shows OJS1[12]; toggles xOJS1[12]
ellipse at (310,100)-(351,141): alarm colour if IN2
ellipse at (480,100)-(521,141): alarm colour if IN3
ellipse at (650,100)-(691,141): alarm colour if IN4
ellipse at (140,260)-(181,301): alarm colour if IN5
ellipse at (310,260)-(351,301): alarm colour if IN6
ellipse at (480,260)-(521,301): alarm colour if IN7
ellipse at (650,260)-(691,301): alarm colour if IN8
ellipse at (140,370)-(181,411): alarm colour if IN9
ellipse at (310,370)-(351,411): alarm colour if IN10
ellipse at (480,370)-(521,411): alarm colour if IN11
ellipse at (650,370)-(691,411): alarm colour if IN12
rectangle at (430,540)-(801,571): text "Stroj má dostatatek materialu na vyrobu"
rectangle at (430,570)-(801,601): text "Stroj ocekava slitinu hliniku"
rectangle at (210,540)-(431,601): text "Filtrovat:"
button at (360,560)-(441,591): text "%s"; shows PLC_PRG.Slitina[1]; opens OJS_I_FS1
button at (270,560)-(351,591): text "Vse"; opens OJS_I
rectangle at (130,60)-(191,181): alarm colour if xOJS1[1]
rectangle at (300,60)-(361,181): alarm colour if xOJS1[2]
rectangle at (470,60)-(531,181): alarm colour if xOJS1[3]
rectangle at (640,60)-(701,181): alarm colour if xOJS1[4]
rectangle at (130,220)-(191,341): alarm colour if xOJS1[5]
rectangle at (300,220)-(361,341): alarm colour if xOJS1[6]
rectangle at (470,220)-(531,341): alarm colour if xOJS1[7]
rectangle at (640,220)-(701,341): alarm colour if xOJS1[8]
rectangle at (130,330)-(191,451): alarm colour if xOJS1[9]
rectangle at (300,330)-(361,451): alarm colour if xOJS1[10]
rectangle at (470,330)-(531,451): alarm colour if xOJS1[11]
rectangle at (640,330)-(701,451): alarm colour if xOJS1[12]
rectangle at (350,0)-(511,41): text "%s"; shows PLC_PRG.Slitina[2]
21 more shapes without text or variables
*)

(* Visualisation OJS1/OJS_I_FS2x
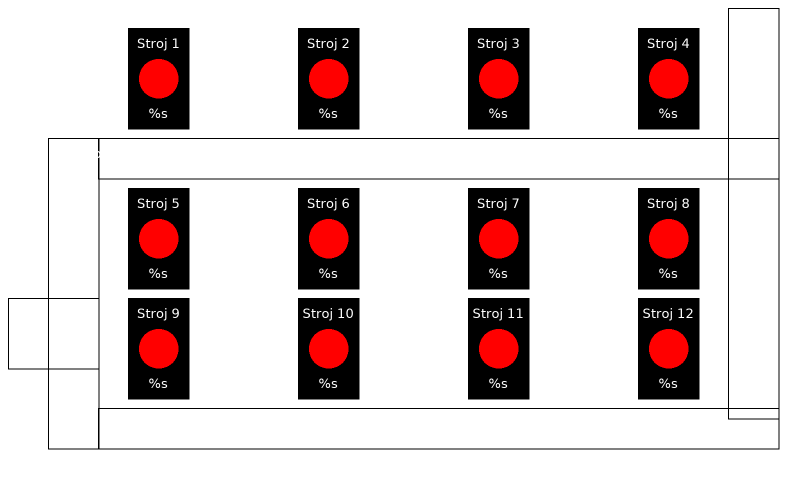
rectangle at (50,130)-(161,161): text "Transportní cesta"
rectangle at (120,20)-(181,51): text "Stroj 1"
ellipse at (130,50)-(171,91): alarm colour if IN1
rectangle at (630,20)-(691,51): text "Stroj 4"
rectangle at (290,20)-(351,51): text "Stroj 2"
rectangle at (460,20)-(521,51): text "Stroj 3"
rectangle at (120,180)-(181,211): text "Stroj 5"
rectangle at (290,180)-(351,211): text "Stroj 6"
rectangle at (460,180)-(521,211): text "Stroj 7"
rectangle at (630,180)-(691,211): text "Stroj 8"
rectangle at (120,290)-(181,321): text "Stroj 9"
rectangle at (290,290)-(351,321): text "Stroj 10"
rectangle at (460,290)-(521,321): text "Stroj 11"
rectangle at (630,290)-(691,321): text "Stroj 12"
rectangle at (120,90)-(181,121): text "%s"; shows OJS1[1]; toggles xOJS1[1]
rectangle at (290,90)-(351,121): text "%s"; shows OJS1[2]; toggles xOJS1[2]
rectangle at (460,90)-(521,121): text "%s"; shows OJS1[3]; toggles xOJS1[3]
rectangle at (630,90)-(691,121): text "%s"; shows OJS1[4]; toggles xOJS1[4]
rectangle at (120,250)-(181,281): text "%s"; shows OJS1[5]; toggles xOJS1[5]
rectangle at (290,250)-(351,281): text "%s"; shows OJS1[6]; toggles xOJS1[6]
rectangle at (460,250)-(521,281): text "%s"; shows OJS1[7]; toggles xOJS1[7]
rectangle at (630,250)-(691,281): text "%s"; shows OJS1[8]; toggles xOJS1[8]
rectangle at (120,360)-(181,391): text "%s"; shows OJS1[9]; toggles xOJS1[9]
rectangle at (290,360)-(351,391): text "%s"; shows OJS1[10]; toggles xOJS1[10]
rectangle at (460,360)-(521,391): text "%s"; shows OJS1[11]; toggles xOJS1[11]
rectangle at (630,360)-(691,391): text "%s"; shows OJS1[12]; toggles xOJS1[12]
ellipse at (300,50)-(341,91): alarm colour if IN2
ellipse at (470,50)-(511,91): alarm colour if IN3
ellipse at (640,50)-(681,91): alarm colour if IN4
ellipse at (130,210)-(171,251): alarm colour if IN5
ellipse at (300,210)-(341,251): alarm colour if IN6
ellipse at (470,210)-(511,251): alarm colour if IN7
ellipse at (640,210)-(681,251): alarm colour if IN8
ellipse at (130,320)-(171,361): alarm colour if IN9
ellipse at (300,320)-(341,361): alarm colour if IN10
ellipse at (470,320)-(511,361): alarm colour if IN11
ellipse at (640,320)-(681,361): alarm colour if IN12
rectangle at (120,10)-(181,131): alarm colour if xOJS1[1]
rectangle at (290,10)-(351,131): alarm colour if xOJS1[2]
rectangle at (460,10)-(521,131): alarm colour if xOJS1[3]
rectangle at (630,10)-(691,131): alarm colour if xOJS1[4]
rectangle at (120,170)-(181,291): alarm colour if xOJS1[5]
rectangle at (290,170)-(351,291): alarm colour if xOJS1[6]
rectangle at (460,170)-(521,291): alarm colour if xOJS1[7]
rectangle at (630,170)-(691,291): alarm colour if xOJS1[8]
rectangle at (120,280)-(181,401): alarm colour if xOJS1[9]
rectangle at (290,280)-(351,401): alarm colour if xOJS1[10]
rectangle at (460,280)-(521,401): alarm colour if xOJS1[11]
rectangle at (630,280)-(691,401): alarm colour if xOJS1[12]
19 more shapes without text or variables
*)

(* Visualisation OJS2/OJS_II
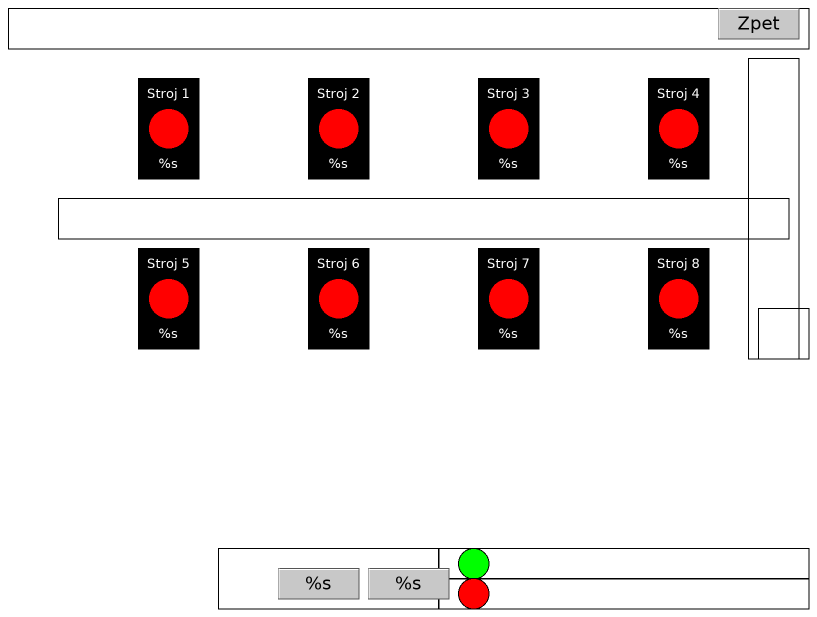
rectangle at (60,140)-(171,171): text "Transportní cesta"
rectangle at (130,240)-(191,271): text "Stroj 5"
rectangle at (300,240)-(361,271): text "Stroj 6"
rectangle at (470,240)-(531,271): text "Stroj 7"
rectangle at (640,240)-(701,271): text "Stroj 8"
rectangle at (640,70)-(701,101): text "Stroj 4"
rectangle at (470,70)-(531,101): text "Stroj 3"
rectangle at (300,70)-(361,101): text "Stroj 2"
rectangle at (130,70)-(191,101): text "Stroj 1"
rectangle at (0,0)-(801,41): text "SLEVARNA AL OJS II"
button at (710,0)-(791,31): text "Zpet"; opens plc_vizu
ellipse at (140,100)-(181,141): alarm colour if Host1IN1
ellipse at (310,100)-(351,141): alarm colour if Host1IN2
ellipse at (480,100)-(521,141): alarm colour if Host1IN3
ellipse at (650,100)-(691,141): alarm colour if Host1IN4
ellipse at (140,270)-(181,311): alarm colour if Host1IN5
ellipse at (310,270)-(351,311): alarm colour if Host1IN6
ellipse at (480,270)-(521,311): alarm colour if Host1IN7
ellipse at (650,270)-(691,311): alarm colour if Host1IN8
rectangle at (130,140)-(191,171): text "%s"; shows OJS2[1]; toggles xOJS2[1]
rectangle at (300,140)-(361,171): text "%s"; shows OJS2[2]; toggles xOJS2[2]
rectangle at (470,140)-(531,171): text "%s"; shows OJS2[3]; toggles xOJS2[3]
rectangle at (640,140)-(701,171): text "%s"; shows OJS2[4]; toggles xOJS2[4]
rectangle at (130,310)-(191,341): text "%s"; shows OJS2[5]; toggles xOJS2[5]
rectangle at (300,310)-(361,341): text "%s"; shows OJS2[6]; toggles xOJS2[6]
rectangle at (470,310)-(531,341): text "%s"; shows OJS2[7]; toggles xOJS2[7]
rectangle at (640,310)-(701,341): text "%s"; shows OJS2[8]; toggles xOJS2[8]
rectangle at (430,540)-(801,571): text "Stroj má dostatatek materialu na vyrobu"
rectangle at (430,570)-(801,601): text "Stroj ocekava slitinu hliniku"
rectangle at (210,540)-(431,601): text "Filtrovat:"
button at (360,560)-(441,591): text "%s"; shows PLC_PRG.Slitina[2]; opens OJS_II_FS2
button at (270,560)-(351,591): text "%s"; shows PLC_PRG.Slitina[1]; opens OJS_II_FS1
15 more shapes without text or variables
*)

(* Visualisation OJS2/OJS_II_FS1
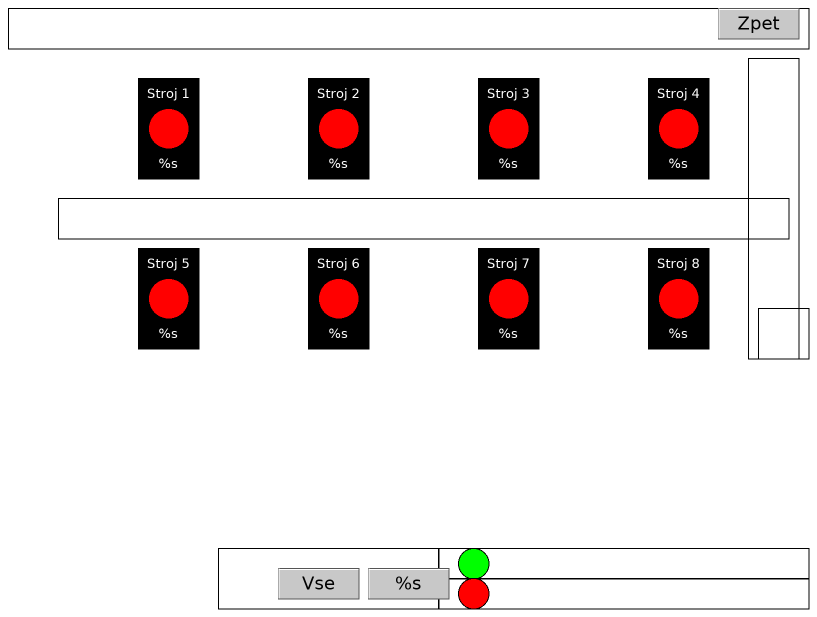
rectangle at (60,140)-(171,171): text "Transportní cesta"
rectangle at (130,240)-(191,271): text "Stroj 5"
rectangle at (300,240)-(361,271): text "Stroj 6"
rectangle at (470,240)-(531,271): text "Stroj 7"
rectangle at (640,240)-(701,271): text "Stroj 8"
rectangle at (640,70)-(701,101): text "Stroj 4"
rectangle at (470,70)-(531,101): text "Stroj 3"
rectangle at (300,70)-(361,101): text "Stroj 2"
rectangle at (130,70)-(191,101): text "Stroj 1"
rectangle at (0,0)-(801,41): text "SLEVARNA AL OJS II - FILTR"
button at (710,0)-(791,31): text "Zpet"; opens plc_vizu
ellipse at (140,100)-(181,141): alarm colour if Host1IN1
ellipse at (310,100)-(351,141): alarm colour if Host1IN2
ellipse at (480,100)-(521,141): alarm colour if Host1IN3
ellipse at (650,100)-(691,141): alarm colour if Host1IN4
ellipse at (140,270)-(181,311): alarm colour if Host1IN5
ellipse at (310,270)-(351,311): alarm colour if Host1IN6
ellipse at (480,270)-(521,311): alarm colour if Host1IN7
ellipse at (650,270)-(691,311): alarm colour if Host1IN8
rectangle at (130,140)-(191,171): text "%s"; shows OJS2[1]; toggles xOJS2[1]
rectangle at (300,140)-(361,171): text "%s"; shows OJS2[2]; toggles xOJS2[2]
rectangle at (470,140)-(531,171): text "%s"; shows OJS2[3]; toggles xOJS2[3]
rectangle at (640,140)-(701,171): text "%s"; shows OJS2[4]; toggles xOJS2[4]
rectangle at (130,310)-(191,341): text "%s"; shows OJS2[5]; toggles xOJS2[5]
rectangle at (300,310)-(361,341): text "%s"; shows OJS2[6]; toggles xOJS2[6]
rectangle at (470,310)-(531,341): text "%s"; shows OJS2[7]; toggles xOJS2[7]
rectangle at (640,310)-(701,341): text "%s"; shows OJS2[8]; toggles xOJS2[8]
rectangle at (430,540)-(801,571): text "Stroj má dostatatek materialu na vyrobu"
rectangle at (430,570)-(801,601): text "Stroj ocekava slitinu hliniku"
rectangle at (210,540)-(431,601): text "Filtrovat:"
button at (360,560)-(441,591): text "%s"; shows PLC_PRG.Slitina[2]; opens OJS_II_FS2
rectangle at (350,0)-(511,41): text "%s"; shows PLC_PRG.Slitina[1]
rectangle at (130,60)-(191,181): alarm colour if xxOJS2[1]
rectangle at (300,60)-(361,181): alarm colour if xxOJS2[2]
rectangle at (470,60)-(531,181): alarm colour if xxOJS2[3]
rectangle at (640,60)-(701,181): alarm colour if xxOJS2[4]
rectangle at (130,230)-(191,351): alarm colour if xxOJS2[5]
rectangle at (300,230)-(361,351): alarm colour if xxOJS2[6]
rectangle at (470,230)-(531,351): alarm colour if xxOJS2[7]
rectangle at (640,230)-(701,351): alarm colour if xxOJS2[8]
button at (270,560)-(351,591): text "Vse"; opens OJS_II
15 more shapes without text or variables
*)

(* Visualisation OJS2/OJS_II_FS1x
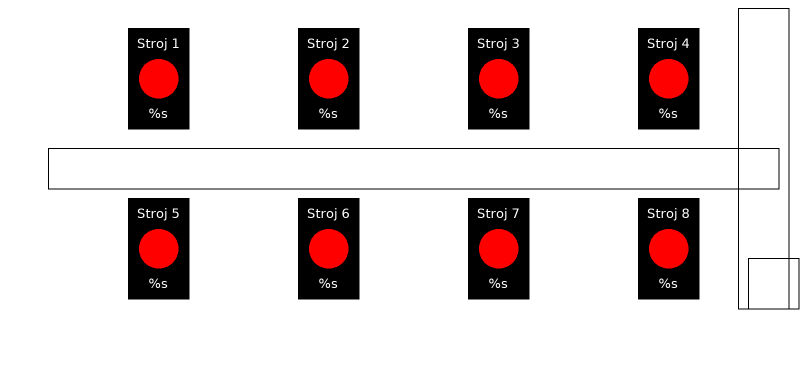
rectangle at (50,90)-(161,121): text "Transportní cesta"
rectangle at (120,190)-(181,221): text "Stroj 5"
rectangle at (290,190)-(351,221): text "Stroj 6"
rectangle at (460,190)-(521,221): text "Stroj 7"
rectangle at (630,190)-(691,221): text "Stroj 8"
rectangle at (630,20)-(691,51): text "Stroj 4"
rectangle at (460,20)-(521,51): text "Stroj 3"
rectangle at (290,20)-(351,51): text "Stroj 2"
rectangle at (120,20)-(181,51): text "Stroj 1"
ellipse at (130,50)-(171,91): alarm colour if Host1IN1
ellipse at (300,50)-(341,91): alarm colour if Host1IN2
ellipse at (470,50)-(511,91): alarm colour if Host1IN3
ellipse at (640,50)-(681,91): alarm colour if Host1IN4
ellipse at (130,220)-(171,261): alarm colour if Host1IN5
ellipse at (300,220)-(341,261): alarm colour if Host1IN6
ellipse at (470,220)-(511,261): alarm colour if Host1IN7
ellipse at (640,220)-(681,261): alarm colour if Host1IN8
rectangle at (120,90)-(181,121): text "%s"; shows OJS2[1]; toggles xOJS2[1]
rectangle at (290,90)-(351,121): text "%s"; shows OJS2[2]; toggles xOJS2[2]
rectangle at (460,90)-(521,121): text "%s"; shows OJS2[3]; toggles xOJS2[3]
rectangle at (630,90)-(691,121): text "%s"; shows OJS2[4]; toggles xOJS2[4]
rectangle at (120,260)-(181,291): text "%s"; shows OJS2[5]; toggles xOJS2[5]
rectangle at (290,260)-(351,291): text "%s"; shows OJS2[6]; toggles xOJS2[6]
rectangle at (460,260)-(521,291): text "%s"; shows OJS2[7]; toggles xOJS2[7]
rectangle at (630,260)-(691,291): text "%s"; shows OJS2[8]; toggles xOJS2[8]
rectangle at (120,10)-(181,131): alarm colour if xxOJS2[1]
rectangle at (290,10)-(351,131): alarm colour if xxOJS2[2]
rectangle at (460,10)-(521,131): alarm colour if xxOJS2[3]
rectangle at (630,10)-(691,131): alarm colour if xxOJS2[4]
rectangle at (120,180)-(181,301): alarm colour if xxOJS2[5]
rectangle at (290,180)-(351,301): alarm colour if xxOJS2[6]
rectangle at (460,180)-(521,301): alarm colour if xxOJS2[7]
rectangle at (630,180)-(691,301): alarm colour if xxOJS2[8]
13 more shapes without text or variables
*)

(* Visualisation OJS2/OJS_II_FS2
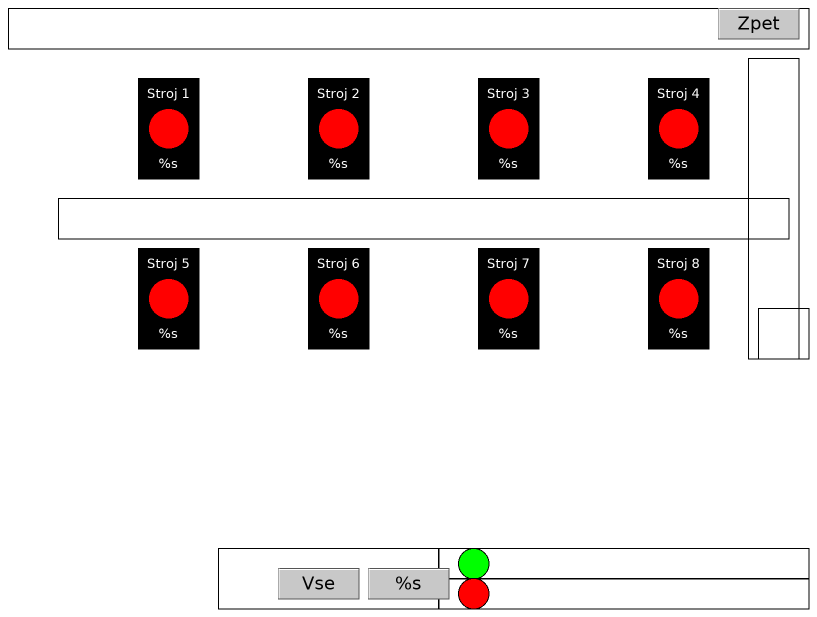
rectangle at (60,140)-(171,171): text "Transportní cesta"
rectangle at (130,240)-(191,271): text "Stroj 5"
rectangle at (300,240)-(361,271): text "Stroj 6"
rectangle at (470,240)-(531,271): text "Stroj 7"
rectangle at (640,240)-(701,271): text "Stroj 8"
rectangle at (640,70)-(701,101): text "Stroj 4"
rectangle at (470,70)-(531,101): text "Stroj 3"
rectangle at (300,70)-(361,101): text "Stroj 2"
rectangle at (130,70)-(191,101): text "Stroj 1"
rectangle at (0,0)-(801,41): text "SLEVARNA AL OJS II - FILTR"
button at (710,0)-(791,31): text "Zpet"; opens plc_vizu
ellipse at (140,100)-(181,141): alarm colour if Host1IN1
ellipse at (310,100)-(351,141): alarm colour if Host1IN2
ellipse at (480,100)-(521,141): alarm colour if Host1IN3
ellipse at (650,100)-(691,141): alarm colour if Host1IN4
ellipse at (140,270)-(181,311): alarm colour if Host1IN5
ellipse at (310,270)-(351,311): alarm colour if Host1IN6
ellipse at (480,270)-(521,311): alarm colour if Host1IN7
ellipse at (650,270)-(691,311): alarm colour if Host1IN8
rectangle at (130,140)-(191,171): text "%s"; shows OJS2[1]; toggles xOJS2[1]
rectangle at (300,140)-(361,171): text "%s"; shows OJS2[2]; toggles xOJS2[2]
rectangle at (470,140)-(531,171): text "%s"; shows OJS2[3]; toggles xOJS2[3]
rectangle at (640,140)-(701,171): text "%s"; shows OJS2[4]; toggles xOJS2[4]
rectangle at (130,310)-(191,341): text "%s"; shows OJS2[5]; toggles xOJS2[5]
rectangle at (300,310)-(361,341): text "%s"; shows OJS2[6]; toggles xOJS2[6]
rectangle at (470,310)-(531,341): text "%s"; shows OJS2[7]; toggles xOJS2[7]
rectangle at (640,310)-(701,341): text "%s"; shows OJS2[8]; toggles xOJS2[8]
rectangle at (430,540)-(801,571): text "Stroj má dostatatek materialu na vyrobu"
rectangle at (430,570)-(801,601): text "Stroj ocekava slitinu hliniku"
rectangle at (210,540)-(431,601): text "Filtrovat:"
button at (360,560)-(441,591): text "%s"; shows PLC_PRG.Slitina[2]; opens OJS_II_FS2
rectangle at (350,0)-(511,41): text "%s"; shows PLC_PRG.Slitina[2]
rectangle at (130,60)-(191,181): alarm colour if xOJS2[1]
rectangle at (300,60)-(361,181): alarm colour if xOJS2[2]
rectangle at (470,60)-(531,181): alarm colour if xOJS2[3]
rectangle at (640,60)-(701,181): alarm colour if xOJS2[4]
rectangle at (130,230)-(191,351): alarm colour if xOJS2[5]
rectangle at (300,230)-(361,351): alarm colour if xOJS2[6]
rectangle at (470,230)-(531,351): alarm colour if xOJS2[7]
rectangle at (640,230)-(701,351): alarm colour if xOJS2[8]
button at (270,560)-(351,591): text "Vse"; opens OJS_II
15 more shapes without text or variables
*)

(* Visualisation OJS2/OJS_II_FS2x
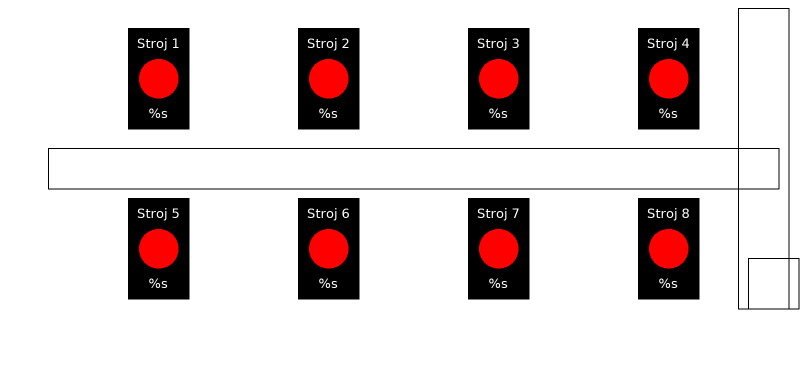
rectangle at (50,90)-(161,121): text "Transportní cesta"
rectangle at (120,190)-(181,221): text "Stroj 5"
rectangle at (290,190)-(351,221): text "Stroj 6"
rectangle at (460,190)-(521,221): text "Stroj 7"
rectangle at (630,190)-(691,221): text "Stroj 8"
rectangle at (630,20)-(691,51): text "Stroj 4"
rectangle at (460,20)-(521,51): text "Stroj 3"
rectangle at (290,20)-(351,51): text "Stroj 2"
rectangle at (120,20)-(181,51): text "Stroj 1"
ellipse at (130,50)-(171,91): alarm colour if Host1IN1
ellipse at (300,50)-(341,91): alarm colour if Host1IN2
ellipse at (470,50)-(511,91): alarm colour if Host1IN3
ellipse at (640,50)-(681,91): alarm colour if Host1IN4
ellipse at (130,220)-(171,261): alarm colour if Host1IN5
ellipse at (300,220)-(341,261): alarm colour if Host1IN6
ellipse at (470,220)-(511,261): alarm colour if Host1IN7
ellipse at (640,220)-(681,261): alarm colour if Host1IN8
rectangle at (120,90)-(181,121): text "%s"; shows OJS2[1]; toggles xOJS2[1]
rectangle at (290,90)-(351,121): text "%s"; shows OJS2[2]; toggles xOJS2[2]
rectangle at (460,90)-(521,121): text "%s"; shows OJS2[3]; toggles xOJS2[3]
rectangle at (630,90)-(691,121): text "%s"; shows OJS2[4]; toggles xOJS2[4]
rectangle at (120,260)-(181,291): text "%s"; shows OJS2[5]; toggles xOJS2[5]
rectangle at (290,260)-(351,291): text "%s"; shows OJS2[6]; toggles xOJS2[6]
rectangle at (460,260)-(521,291): text "%s"; shows OJS2[7]; toggles xOJS2[7]
rectangle at (630,260)-(691,291): text "%s"; shows OJS2[8]; toggles xOJS2[8]
rectangle at (120,10)-(181,131): alarm colour if xOJS2[1]
rectangle at (290,10)-(351,131): alarm colour if xOJS2[2]
rectangle at (460,10)-(521,131): alarm colour if xOJS2[3]
rectangle at (630,10)-(691,131): alarm colour if xOJS2[4]
rectangle at (120,180)-(181,301): alarm colour if xOJS2[5]
rectangle at (290,180)-(351,301): alarm colour if xOJS2[6]
rectangle at (460,180)-(521,301): alarm colour if xOJS2[7]
rectangle at (630,180)-(691,301): alarm colour if xOJS2[8]
13 more shapes without text or variables
*)

(* Visualisation OJS3/OJS_III
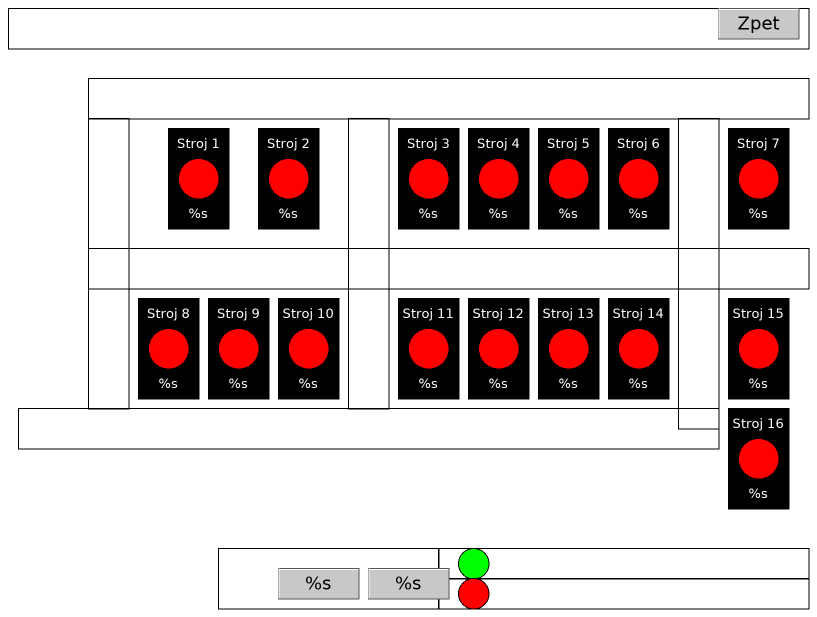
rectangle at (90,70)-(201,101): text "Transportní cesta"
rectangle at (430,120)-(551,151): text "Stroj 4"
rectangle at (600,120)-(661,151): text "Stroj 6"
rectangle at (530,120)-(591,151): text "Stroj 5"
rectangle at (390,120)-(451,151): text "Stroj 3"
rectangle at (720,120)-(781,151): text "Stroj 7"
rectangle at (250,120)-(311,151): text "Stroj 2"
rectangle at (160,120)-(221,151): text "Stroj 1"
rectangle at (600,290)-(661,321): text "Stroj 14"
rectangle at (530,290)-(591,321): text "Stroj 13"
rectangle at (390,290)-(451,321): text "Stroj 11"
rectangle at (720,290)-(781,321): text "Stroj 15"
rectangle at (720,400)-(781,431): text "Stroj 16"
rectangle at (270,290)-(331,321): text "Stroj 10"
rectangle at (200,290)-(261,321): text "Stroj 9"
rectangle at (130,290)-(191,321): text "Stroj 8"
rectangle at (460,290)-(521,321): text "Stroj 12"
rectangle at (0,0)-(801,41): text "SLEVARNA AL OJS III"
button at (710,0)-(791,31): text "Zpet"; opens plc_vizu
rectangle at (430,540)-(801,571): text "Stroj má dostatatek materialu na vyrobu"
rectangle at (430,570)-(801,601): text "Stroj ocekava slitinu hliniku"
rectangle at (160,190)-(221,221): text "%s"; shows OJS3[1]; toggles xOJS3[1]
ellipse at (170,150)-(211,191): alarm colour if Host2IN1
ellipse at (260,150)-(301,191): alarm colour if Host2IN2
ellipse at (400,150)-(441,191): alarm colour if Host2IN3
ellipse at (470,150)-(511,191): alarm colour if Host2IN4
ellipse at (540,150)-(581,191): alarm colour if Host2IN5
ellipse at (610,150)-(651,191): alarm colour if Host2IN6
ellipse at (730,150)-(771,191): alarm colour if Host2IN7
ellipse at (140,320)-(181,361): alarm colour if Host2IN8
ellipse at (210,320)-(251,361): alarm colour if Host2IN9
ellipse at (280,320)-(321,361): alarm colour if Host2IN10
ellipse at (400,320)-(441,361): alarm colour if Host2IN11
ellipse at (470,320)-(511,361): alarm colour if Host2IN12
ellipse at (540,320)-(581,361): alarm colour if Host2IN13
ellipse at (610,320)-(651,361): alarm colour if Host2IN14
ellipse at (730,320)-(771,361): alarm colour if Host2IN15
ellipse at (730,430)-(771,471): alarm colour if Host2IN16
rectangle at (250,190)-(311,221): text "%s"; shows OJS3[2]; toggles xOJS3[2]
rectangle at (390,190)-(451,221): text "%s"; shows OJS3[3]; toggles xOJS3[3]
rectangle at (460,190)-(521,221): text "%s"; shows OJS3[4]; toggles xOJS3[4]
rectangle at (530,190)-(591,221): text "%s"; shows OJS3[5]; toggles xOJS3[5]
rectangle at (600,190)-(661,221): text "%s"; shows OJS3[6]; toggles xOJS3[6]
rectangle at (720,190)-(781,221): text "%s"; shows OJS3[7]; toggles xOJS3[7]
rectangle at (130,360)-(191,391): text "%s"; shows OJS3[8]; toggles xOJS3[8]
rectangle at (200,360)-(261,391): text "%s"; shows OJS3[9]; toggles xOJS3[9]
rectangle at (270,360)-(331,391): text "%s"; shows OJS3[10]; toggles xOJS3[10]
rectangle at (390,360)-(451,391): text "%s"; shows OJS3[11]; toggles xOJS3[11]
rectangle at (460,360)-(521,391): text "%s"; shows OJS3[12]; toggles xOJS3[12]
rectangle at (530,360)-(591,391): text "%s"; shows OJS3[13]; toggles xOJS3[13]
rectangle at (600,360)-(661,391): text "%s"; shows OJS3[14]; toggles xOJS3[14]
rectangle at (720,360)-(781,391): text "%s"; shows OJS3[15]; toggles xOJS3[15]
rectangle at (720,470)-(781,501): text "%s"; shows OJS3[16]; toggles xOJS3[16]
rectangle at (210,540)-(431,601): text "Filtrovat:"
button at (360,560)-(441,591): text "%s"; shows PLC_PRG.Slitina[2]; opens OJS_III_FS2
button at (270,560)-(351,591): text "%s"; shows PLC_PRG.Slitina[1]; opens OJS_III_FS1
26 more shapes without text or variables
*)

(* Visualisation OJS3/OJS_III_FS1
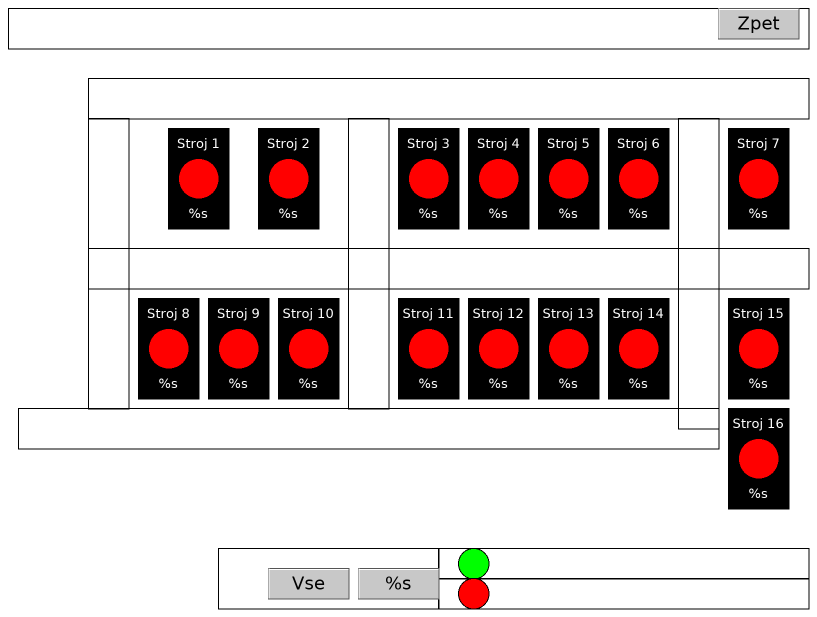
rectangle at (90,70)-(201,101): text "Transportní cesta"
rectangle at (430,120)-(551,151): text "Stroj 4"
rectangle at (600,120)-(661,151): text "Stroj 6"
rectangle at (530,120)-(591,151): text "Stroj 5"
rectangle at (390,120)-(451,151): text "Stroj 3"
rectangle at (720,120)-(781,151): text "Stroj 7"
rectangle at (250,120)-(311,151): text "Stroj 2"
rectangle at (160,120)-(221,151): text "Stroj 1"
rectangle at (600,290)-(661,321): text "Stroj 14"
rectangle at (530,290)-(591,321): text "Stroj 13"
rectangle at (390,290)-(451,321): text "Stroj 11"
rectangle at (720,290)-(781,321): text "Stroj 15"
rectangle at (720,400)-(781,431): text "Stroj 16"
rectangle at (270,290)-(331,321): text "Stroj 10"
rectangle at (200,290)-(261,321): text "Stroj 9"
rectangle at (130,290)-(191,321): text "Stroj 8"
rectangle at (460,290)-(521,321): text "Stroj 12"
rectangle at (0,0)-(801,41): text "SLEVARNA AL OJS III - FILTR"
button at (710,0)-(791,31): text "Zpet"; opens plc_vizu
rectangle at (430,540)-(801,571): text "Stroj má dostatatek materialu na vyrobu"
rectangle at (430,570)-(801,601): text "Stroj ocekava slitinu hliniku"
rectangle at (160,190)-(221,221): text "%s"; shows OJS3[1]; toggles xOJS3[1]
ellipse at (170,150)-(211,191): alarm colour if Host2IN1
ellipse at (260,150)-(301,191): alarm colour if Host2IN2
ellipse at (400,150)-(441,191): alarm colour if Host2IN3
ellipse at (470,150)-(511,191): alarm colour if Host2IN4
ellipse at (540,150)-(581,191): alarm colour if Host2IN5
ellipse at (610,150)-(651,191): alarm colour if Host2IN6
ellipse at (730,150)-(771,191): alarm colour if Host2IN7
ellipse at (140,320)-(181,361): alarm colour if Host2IN8
ellipse at (210,320)-(251,361): alarm colour if Host2IN9
ellipse at (280,320)-(321,361): alarm colour if Host2IN10
ellipse at (400,320)-(441,361): alarm colour if Host2IN11
ellipse at (470,320)-(511,361): alarm colour if Host2IN12
ellipse at (540,320)-(581,361): alarm colour if Host2IN13
ellipse at (610,320)-(651,361): alarm colour if Host2IN14
ellipse at (730,320)-(771,361): alarm colour if Host2IN15
ellipse at (730,430)-(771,471): alarm colour if Host2IN16
rectangle at (250,190)-(311,221): text "%s"; shows OJS3[2]; toggles xOJS3[2]
rectangle at (390,190)-(451,221): text "%s"; shows OJS3[3]; toggles xOJS3[3]
rectangle at (460,190)-(521,221): text "%s"; shows OJS3[4]; toggles xOJS3[4]
rectangle at (530,190)-(591,221): text "%s"; shows OJS3[5]; toggles xOJS3[5]
rectangle at (600,190)-(661,221): text "%s"; shows OJS3[6]; toggles xOJS3[6]
rectangle at (720,190)-(781,221): text "%s"; shows OJS3[7]; toggles xOJS3[7]
rectangle at (130,360)-(191,391): text "%s"; shows OJS3[8]; toggles xOJS3[8]
rectangle at (200,360)-(261,391): text "%s"; shows OJS3[9]; toggles xOJS3[9]
rectangle at (270,360)-(331,391): text "%s"; shows OJS3[10]; toggles xOJS3[10]
rectangle at (390,360)-(451,391): text "%s"; shows OJS3[11]; toggles xOJS3[11]
rectangle at (460,360)-(521,391): text "%s"; shows OJS3[12]; toggles xOJS3[12]
rectangle at (530,360)-(591,391): text "%s"; shows OJS3[13]; toggles xOJS3[13]
rectangle at (600,360)-(661,391): text "%s"; shows OJS3[14]; toggles xOJS3[14]
rectangle at (720,360)-(781,391): text "%s"; shows OJS3[15]; toggles xOJS3[15]
rectangle at (720,470)-(781,501): text "%s"; shows OJS3[16]; toggles xOJS3[16]
rectangle at (210,540)-(431,601): text "Filtrovat:"
button at (350,560)-(431,591): text "%s"; shows PLC_PRG.Slitina[2]; opens OJS_III_FS2
rectangle at (360,0)-(521,41): text "%s"; shows PLC_PRG.Slitina[1]
rectangle at (160,110)-(221,231): alarm colour if xxOJS3[1]
rectangle at (250,110)-(311,231): alarm colour if xxOJS3[2]
rectangle at (390,110)-(451,231): alarm colour if xxOJS3[3]
rectangle at (460,110)-(521,231): alarm colour if xxOJS3[4]
rectangle at (530,110)-(591,231): alarm colour if xxOJS3[5]
rectangle at (600,110)-(661,231): alarm colour if xxOJS3[6]
rectangle at (720,110)-(781,231): alarm colour if xxOJS3[7]
rectangle at (130,280)-(191,401): alarm colour if xxOJS3[8]
rectangle at (200,280)-(261,401): alarm colour if xxOJS3[9]
rectangle at (270,280)-(331,401): alarm colour if xxOJS3[10]
rectangle at (390,280)-(451,401): alarm colour if xxOJS3[11]
rectangle at (460,280)-(521,401): alarm colour if xxOJS3[12]
rectangle at (530,280)-(591,401): alarm colour if xxOJS3[13]
rectangle at (600,280)-(661,401): alarm colour if xxOJS3[14]
rectangle at (720,280)-(781,401): alarm colour if xxOJS3[15]
rectangle at (720,390)-(781,501): alarm colour if xxOJS3[16]
button at (260,560)-(341,591): text "Vse"; opens OJS_III
26 more shapes without text or variables
*)

(* Visualisation OJS3/OJS_III_FS1x
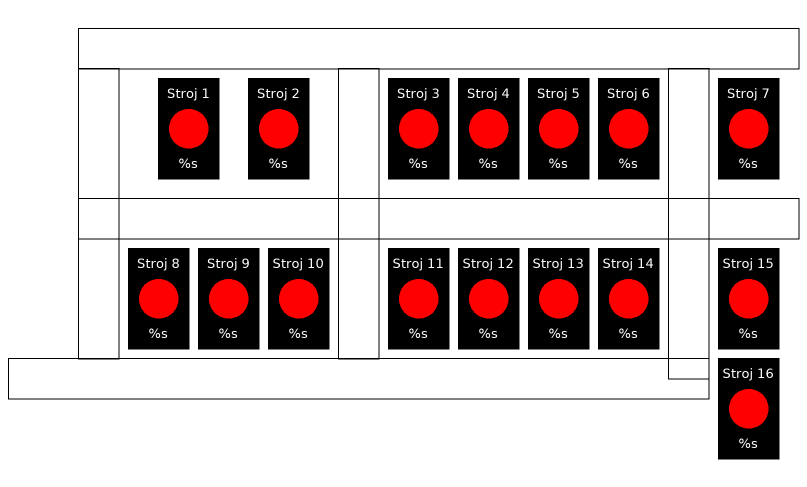
rectangle at (80,20)-(191,51): text "Transportní cesta"
rectangle at (420,70)-(541,101): text "Stroj 4"
rectangle at (590,70)-(651,101): text "Stroj 6"
rectangle at (520,70)-(581,101): text "Stroj 5"
rectangle at (380,70)-(441,101): text "Stroj 3"
rectangle at (710,70)-(771,101): text "Stroj 7"
rectangle at (240,70)-(301,101): text "Stroj 2"
rectangle at (150,70)-(211,101): text "Stroj 1"
rectangle at (590,240)-(651,271): text "Stroj 14"
rectangle at (520,240)-(581,271): text "Stroj 13"
rectangle at (380,240)-(441,271): text "Stroj 11"
rectangle at (710,240)-(771,271): text "Stroj 15"
rectangle at (710,350)-(771,381): text "Stroj 16"
rectangle at (260,240)-(321,271): text "Stroj 10"
rectangle at (190,240)-(251,271): text "Stroj 9"
rectangle at (120,240)-(181,271): text "Stroj 8"
rectangle at (450,240)-(511,271): text "Stroj 12"
rectangle at (150,140)-(211,171): text "%s"; shows OJS3[1]; toggles xOJS3[1]
ellipse at (160,100)-(201,141): alarm colour if Host2IN1
ellipse at (250,100)-(291,141): alarm colour if Host2IN2
ellipse at (390,100)-(431,141): alarm colour if Host2IN3
ellipse at (460,100)-(501,141): alarm colour if Host2IN4
ellipse at (530,100)-(571,141): alarm colour if Host2IN5
ellipse at (600,100)-(641,141): alarm colour if Host2IN6
ellipse at (720,100)-(761,141): alarm colour if Host2IN7
ellipse at (130,270)-(171,311): alarm colour if Host2IN8
ellipse at (200,270)-(241,311): alarm colour if Host2IN9
ellipse at (270,270)-(311,311): alarm colour if Host2IN10
ellipse at (390,270)-(431,311): alarm colour if Host2IN11
ellipse at (460,270)-(501,311): alarm colour if Host2IN12
ellipse at (530,270)-(571,311): alarm colour if Host2IN13
ellipse at (600,270)-(641,311): alarm colour if Host2IN14
ellipse at (720,270)-(761,311): alarm colour if Host2IN15
ellipse at (720,380)-(761,421): alarm colour if Host2IN16
rectangle at (240,140)-(301,171): text "%s"; shows OJS3[2]; toggles xOJS3[2]
rectangle at (380,140)-(441,171): text "%s"; shows OJS3[3]; toggles xOJS3[3]
rectangle at (450,140)-(511,171): text "%s"; shows OJS3[4]; toggles xOJS3[4]
rectangle at (520,140)-(581,171): text "%s"; shows OJS3[5]; toggles xOJS3[5]
rectangle at (590,140)-(651,171): text "%s"; shows OJS3[6]; toggles xOJS3[6]
rectangle at (710,140)-(771,171): text "%s"; shows OJS3[7]; toggles xOJS3[7]
rectangle at (120,310)-(181,341): text "%s"; shows OJS3[8]; toggles xOJS3[8]
rectangle at (190,310)-(251,341): text "%s"; shows OJS3[9]; toggles xOJS3[9]
rectangle at (260,310)-(321,341): text "%s"; shows OJS3[10]; toggles xOJS3[10]
rectangle at (380,310)-(441,341): text "%s"; shows OJS3[11]; toggles xOJS3[11]
rectangle at (450,310)-(511,341): text "%s"; shows OJS3[12]; toggles xOJS3[12]
rectangle at (520,310)-(581,341): text "%s"; shows OJS3[13]; toggles xOJS3[13]
rectangle at (590,310)-(651,341): text "%s"; shows OJS3[14]; toggles xOJS3[14]
rectangle at (710,310)-(771,341): text "%s"; shows OJS3[15]; toggles xOJS3[15]
rectangle at (710,420)-(771,451): text "%s"; shows OJS3[16]; toggles xOJS3[16]
rectangle at (150,60)-(211,181): alarm colour if xxOJS3[1]
rectangle at (240,60)-(301,181): alarm colour if xxOJS3[2]
rectangle at (380,60)-(441,181): alarm colour if xxOJS3[3]
rectangle at (450,60)-(511,181): alarm colour if xxOJS3[4]
rectangle at (520,60)-(581,181): alarm colour if xxOJS3[5]
rectangle at (590,60)-(651,181): alarm colour if xxOJS3[6]
rectangle at (710,60)-(771,181): alarm colour if xxOJS3[7]
rectangle at (120,230)-(181,351): alarm colour if xxOJS3[8]
rectangle at (190,230)-(251,351): alarm colour if xxOJS3[9]
rectangle at (260,230)-(321,351): alarm colour if xxOJS3[10]
rectangle at (380,230)-(441,351): alarm colour if xxOJS3[11]
rectangle at (450,230)-(511,351): alarm colour if xxOJS3[12]
rectangle at (520,230)-(581,351): alarm colour if xxOJS3[13]
rectangle at (590,230)-(651,351): alarm colour if xxOJS3[14]
rectangle at (710,230)-(771,351): alarm colour if xxOJS3[15]
rectangle at (710,340)-(771,451): alarm colour if xxOJS3[16]
24 more shapes without text or variables
*)

(* Visualisation OJS3/OJS_III_FS2
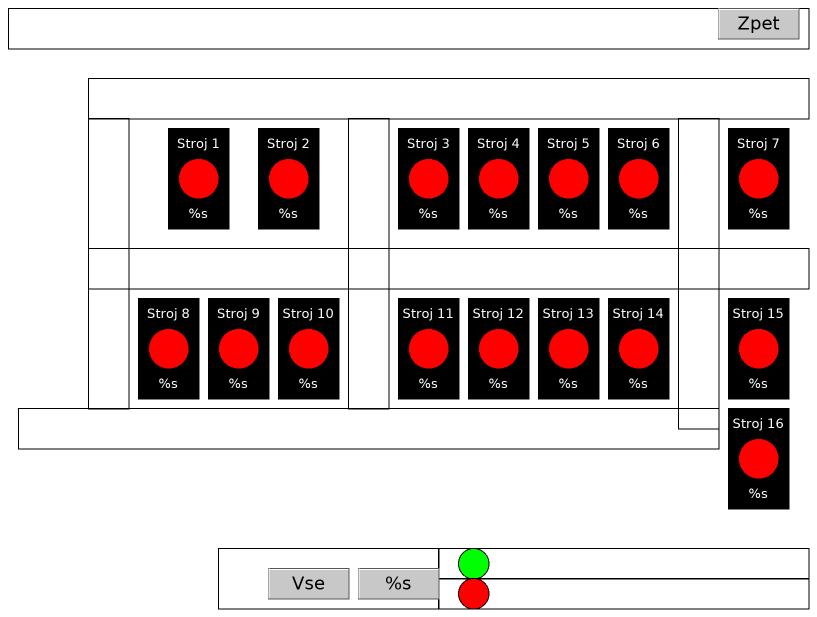
rectangle at (90,70)-(201,101): text "Transportní cesta"
rectangle at (430,120)-(551,151): text "Stroj 4"
rectangle at (600,120)-(661,151): text "Stroj 6"
rectangle at (530,120)-(591,151): text "Stroj 5"
rectangle at (390,120)-(451,151): text "Stroj 3"
rectangle at (720,120)-(781,151): text "Stroj 7"
rectangle at (250,120)-(311,151): text "Stroj 2"
rectangle at (160,120)-(221,151): text "Stroj 1"
rectangle at (600,290)-(661,321): text "Stroj 14"
rectangle at (530,290)-(591,321): text "Stroj 13"
rectangle at (390,290)-(451,321): text "Stroj 11"
rectangle at (720,290)-(781,321): text "Stroj 15"
rectangle at (720,400)-(781,431): text "Stroj 16"
rectangle at (270,290)-(331,321): text "Stroj 10"
rectangle at (200,290)-(261,321): text "Stroj 9"
rectangle at (130,290)-(191,321): text "Stroj 8"
rectangle at (460,290)-(521,321): text "Stroj 12"
rectangle at (0,0)-(801,41): text "SLEVARNA AL OJS III - FILTR"
button at (710,0)-(791,31): text "Zpet"; opens plc_vizu
rectangle at (430,540)-(801,571): text "Stroj má dostatatek materialu na vyrobu"
rectangle at (430,570)-(801,601): text "Stroj ocekava slitinu hliniku"
rectangle at (160,190)-(221,221): text "%s"; shows OJS3[1]; toggles xOJS3[1]
ellipse at (170,150)-(211,191): alarm colour if Host2IN1
ellipse at (260,150)-(301,191): alarm colour if Host2IN2
ellipse at (400,150)-(441,191): alarm colour if Host2IN3
ellipse at (470,150)-(511,191): alarm colour if Host2IN4
ellipse at (540,150)-(581,191): alarm colour if Host2IN5
ellipse at (610,150)-(651,191): alarm colour if Host2IN6
ellipse at (730,150)-(771,191): alarm colour if Host2IN7
ellipse at (140,320)-(181,361): alarm colour if Host2IN8
ellipse at (210,320)-(251,361): alarm colour if Host2IN9
ellipse at (280,320)-(321,361): alarm colour if Host2IN10
ellipse at (400,320)-(441,361): alarm colour if Host2IN11
ellipse at (470,320)-(511,361): alarm colour if Host2IN12
ellipse at (540,320)-(581,361): alarm colour if Host2IN13
ellipse at (610,320)-(651,361): alarm colour if Host2IN14
ellipse at (730,320)-(771,361): alarm colour if Host2IN15
ellipse at (730,430)-(771,471): alarm colour if Host2IN16
rectangle at (250,190)-(311,221): text "%s"; shows OJS3[2]; toggles xOJS3[2]
rectangle at (390,190)-(451,221): text "%s"; shows OJS3[3]; toggles xOJS3[3]
rectangle at (460,190)-(521,221): text "%s"; shows OJS3[4]; toggles xOJS3[4]
rectangle at (530,190)-(591,221): text "%s"; shows OJS3[5]; toggles xOJS3[5]
rectangle at (600,190)-(661,221): text "%s"; shows OJS3[6]; toggles xOJS3[6]
rectangle at (720,190)-(781,221): text "%s"; shows OJS3[7]; toggles xOJS3[7]
rectangle at (130,360)-(191,391): text "%s"; shows OJS3[8]; toggles xOJS3[8]
rectangle at (200,360)-(261,391): text "%s"; shows OJS3[9]; toggles xOJS3[9]
rectangle at (270,360)-(331,391): text "%s"; shows OJS3[10]; toggles xOJS3[10]
rectangle at (390,360)-(451,391): text "%s"; shows OJS3[11]; toggles xOJS3[11]
rectangle at (460,360)-(521,391): text "%s"; shows OJS3[12]; toggles xOJS3[12]
rectangle at (530,360)-(591,391): text "%s"; shows OJS3[13]; toggles xOJS3[13]
rectangle at (600,360)-(661,391): text "%s"; shows OJS3[14]; toggles xOJS3[14]
rectangle at (720,360)-(781,391): text "%s"; shows OJS3[15]; toggles xOJS3[15]
rectangle at (720,470)-(781,501): text "%s"; shows OJS3[16]; toggles xOJS3[16]
rectangle at (210,540)-(431,601): text "Filtrovat:"
button at (350,560)-(431,591): text "%s"; shows PLC_PRG.Slitina[1]; opens OJS_III_FS1
rectangle at (360,0)-(521,41): text "%s"; shows PLC_PRG.Slitina[2]
rectangle at (160,110)-(221,231): alarm colour if xOJS3[1]
rectangle at (250,110)-(311,231): alarm colour if xOJS3[2]
rectangle at (390,110)-(451,231): alarm colour if xOJS3[3]
rectangle at (460,110)-(521,231): alarm colour if xOJS3[4]
rectangle at (530,110)-(591,231): alarm colour if xOJS3[5]
rectangle at (600,110)-(661,231): alarm colour if xOJS3[6]
rectangle at (720,110)-(781,231): alarm colour if xOJS3[7]
rectangle at (130,280)-(191,401): alarm colour if xOJS3[8]
rectangle at (200,280)-(261,401): alarm colour if xOJS3[9]
rectangle at (270,280)-(331,401): alarm colour if xOJS3[10]
rectangle at (390,280)-(451,401): alarm colour if xOJS3[11]
rectangle at (460,280)-(521,401): alarm colour if xOJS3[12]
rectangle at (530,280)-(591,401): alarm colour if xOJS3[13]
rectangle at (600,280)-(661,401): alarm colour if xOJS3[14]
rectangle at (720,280)-(781,401): alarm colour if xOJS3[15]
rectangle at (720,390)-(781,501): alarm colour if xOJS3[16]
button at (260,560)-(341,591): text "Vse"; opens OJS_III
26 more shapes without text or variables
*)

(* Visualisation OJS3/OJS_III_FS2x
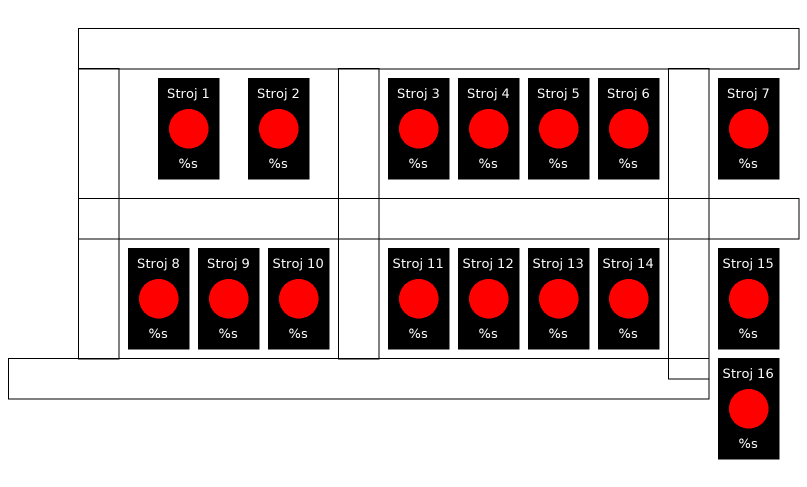
rectangle at (80,20)-(191,51): text "Transportní cesta"
rectangle at (420,70)-(541,101): text "Stroj 4"
rectangle at (590,70)-(651,101): text "Stroj 6"
rectangle at (520,70)-(581,101): text "Stroj 5"
rectangle at (380,70)-(441,101): text "Stroj 3"
rectangle at (710,70)-(771,101): text "Stroj 7"
rectangle at (240,70)-(301,101): text "Stroj 2"
rectangle at (150,70)-(211,101): text "Stroj 1"
rectangle at (590,240)-(651,271): text "Stroj 14"
rectangle at (520,240)-(581,271): text "Stroj 13"
rectangle at (380,240)-(441,271): text "Stroj 11"
rectangle at (710,240)-(771,271): text "Stroj 15"
rectangle at (710,350)-(771,381): text "Stroj 16"
rectangle at (260,240)-(321,271): text "Stroj 10"
rectangle at (190,240)-(251,271): text "Stroj 9"
rectangle at (120,240)-(181,271): text "Stroj 8"
rectangle at (450,240)-(511,271): text "Stroj 12"
rectangle at (150,140)-(211,171): text "%s"; shows OJS3[1]; toggles xOJS3[1]
ellipse at (160,100)-(201,141): alarm colour if Host2IN1
ellipse at (250,100)-(291,141): alarm colour if Host2IN2
ellipse at (390,100)-(431,141): alarm colour if Host2IN3
ellipse at (460,100)-(501,141): alarm colour if Host2IN4
ellipse at (530,100)-(571,141): alarm colour if Host2IN5
ellipse at (600,100)-(641,141): alarm colour if Host2IN6
ellipse at (720,100)-(761,141): alarm colour if Host2IN7
ellipse at (130,270)-(171,311): alarm colour if Host2IN8
ellipse at (200,270)-(241,311): alarm colour if Host2IN9
ellipse at (270,270)-(311,311): alarm colour if Host2IN10
ellipse at (390,270)-(431,311): alarm colour if Host2IN11
ellipse at (460,270)-(501,311): alarm colour if Host2IN12
ellipse at (530,270)-(571,311): alarm colour if Host2IN13
ellipse at (600,270)-(641,311): alarm colour if Host2IN14
ellipse at (720,270)-(761,311): alarm colour if Host2IN15
ellipse at (720,380)-(761,421): alarm colour if Host2IN16
rectangle at (240,140)-(301,171): text "%s"; shows OJS3[2]; toggles xOJS3[2]
rectangle at (380,140)-(441,171): text "%s"; shows OJS3[3]; toggles xOJS3[3]
rectangle at (450,140)-(511,171): text "%s"; shows OJS3[4]; toggles xOJS3[4]
rectangle at (520,140)-(581,171): text "%s"; shows OJS3[5]; toggles xOJS3[5]
rectangle at (590,140)-(651,171): text "%s"; shows OJS3[6]; toggles xOJS3[6]
rectangle at (710,140)-(771,171): text "%s"; shows OJS3[7]; toggles xOJS3[7]
rectangle at (120,310)-(181,341): text "%s"; shows OJS3[8]; toggles xOJS3[8]
rectangle at (190,310)-(251,341): text "%s"; shows OJS3[9]; toggles xOJS3[9]
rectangle at (260,310)-(321,341): text "%s"; shows OJS3[10]; toggles xOJS3[10]
rectangle at (380,310)-(441,341): text "%s"; shows OJS3[11]; toggles xOJS3[11]
rectangle at (450,310)-(511,341): text "%s"; shows OJS3[12]; toggles xOJS3[12]
rectangle at (520,310)-(581,341): text "%s"; shows OJS3[13]; toggles xOJS3[13]
rectangle at (590,310)-(651,341): text "%s"; shows OJS3[14]; toggles xOJS3[14]
rectangle at (710,310)-(771,341): text "%s"; shows OJS3[15]; toggles xOJS3[15]
rectangle at (710,420)-(771,451): text "%s"; shows OJS3[16]; toggles xOJS3[16]
rectangle at (150,60)-(211,181): alarm colour if xOJS3[1]
rectangle at (240,60)-(301,181): alarm colour if xOJS3[2]
rectangle at (380,60)-(441,181): alarm colour if xOJS3[3]
rectangle at (450,60)-(511,181): alarm colour if xOJS3[4]
rectangle at (520,60)-(581,181): alarm colour if xOJS3[5]
rectangle at (590,60)-(651,181): alarm colour if xOJS3[6]
rectangle at (710,60)-(771,181): alarm colour if xOJS3[7]
rectangle at (120,230)-(181,351): alarm colour if xOJS3[8]
rectangle at (190,230)-(251,351): alarm colour if xOJS3[9]
rectangle at (260,230)-(321,351): alarm colour if xOJS3[10]
rectangle at (380,230)-(441,351): alarm colour if xOJS3[11]
rectangle at (450,230)-(511,351): alarm colour if xOJS3[12]
rectangle at (520,230)-(581,351): alarm colour if xOJS3[13]
rectangle at (590,230)-(651,351): alarm colour if xOJS3[14]
rectangle at (710,230)-(771,351): alarm colour if xOJS3[15]
rectangle at (710,340)-(771,451): alarm colour if xOJS3[16]
24 more shapes without text or variables
*)

(* Visualisation plc_vizu
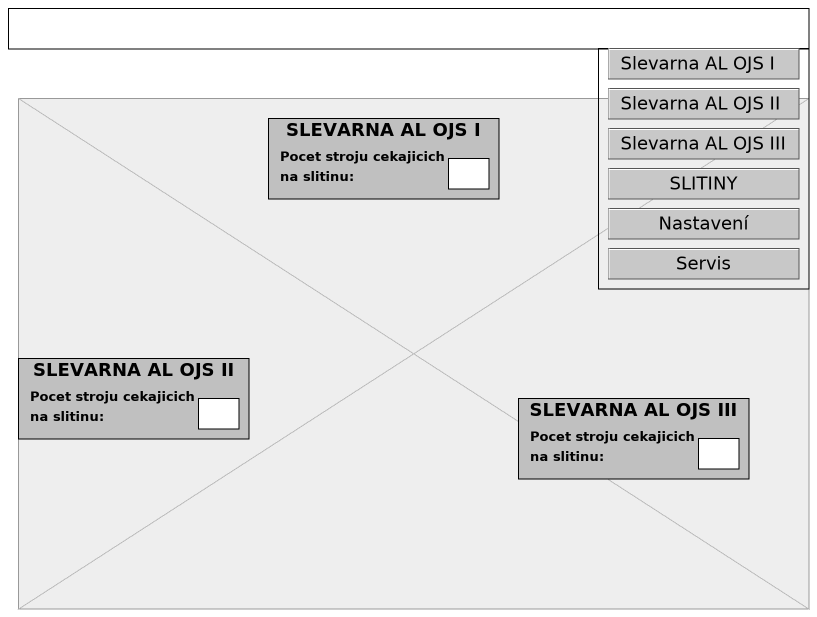
bitmap at (10,90)-(801,601): y:\documents\wago\jhv kovolis hedvikovice\main.bmp
rounded rectangle at (260,110)-(491,191): text "SLEVARNA AL OJS I"; opens OJS_I
rectangle at (0,0)-(801,41): text "KOVOLIS HEDVIKOV"
button at (600,240)-(791,271): text "Servis"; opens Servis
button at (600,200)-(791,231): text "Nastavení"; opens Nastaveni
button at (600,40)-(791,71): text "Slevarna AL OJS I"; opens OJS_I
button at (600,80)-(791,111): text "Slevarna AL OJS II"; opens OJS_II
button at (600,120)-(791,151): text "Slevarna AL OJS III"; opens OJS_III
rectangle at (270,140)-(491,161): text "Pocet stroju cekajicich"; opens OJS_I
rectangle at (270,160)-(491,181): text "na slitinu:"; opens OJS_I
rounded rectangle at (440,150)-(481,181): opens OJS_I
rounded rectangle at (10,350)-(241,431): text "SLEVARNA AL OJS II"; opens OJS_II
rectangle at (20,380)-(241,401): text "Pocet stroju cekajicich"; opens OJS_II
rectangle at (20,400)-(241,421): text "na slitinu:"; opens OJS_II
rounded rectangle at (190,390)-(231,421): opens OJS_II
rounded rectangle at (510,390)-(741,471): text "SLEVARNA AL OJS III"; opens OJS_III
rectangle at (520,420)-(741,441): text "Pocet stroju cekajicich"; opens OJS_III
rectangle at (520,440)-(741,461): text "na slitinu:"; opens OJS_III
rounded rectangle at (690,430)-(731,461): opens OJS_III
button at (600,160)-(791,191): text "SLITINY"; opens Nastaveni
1 more shapes without text or variables
*)

(* Visualisation Servis
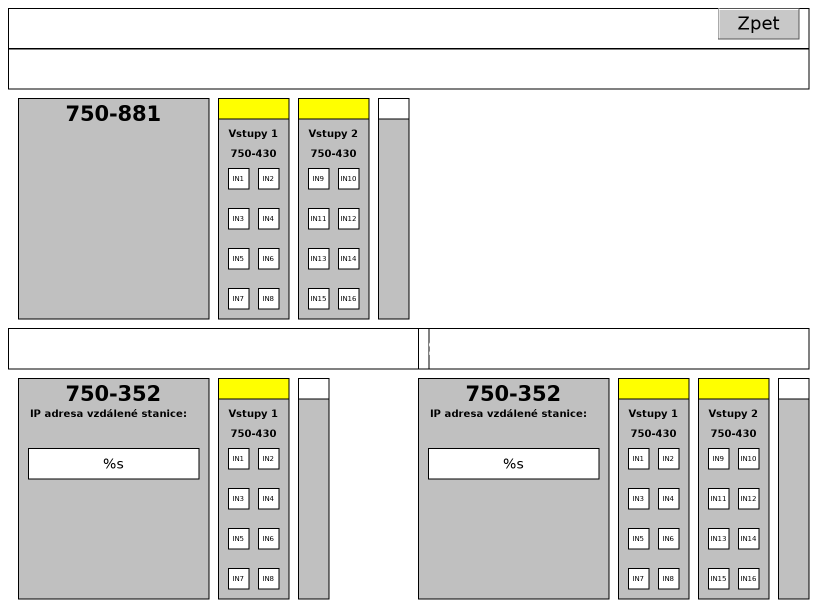
rectangle at (0,0)-(801,41): text "SERVIS"
rectangle at (220,160)-(241,181): text "IN1"; alarm colour if IN1
rectangle at (210,110)-(281,141): text "Vstupy 1"
rectangle at (250,160)-(271,181): text "IN2"; alarm colour if IN2
rectangle at (210,130)-(281,161): text "750-430"
rectangle at (10,90)-(201,121): text "750-881"
rectangle at (220,200)-(241,221): text "IN3"; alarm colour if IN3
rectangle at (250,200)-(271,221): text "IN4"; alarm colour if IN4
rectangle at (220,240)-(241,261): text "IN5"; alarm colour if IN5
rectangle at (250,240)-(271,261): text "IN6"; alarm colour if IN6
rectangle at (220,280)-(241,301): text "IN7"; alarm colour if IN7
rectangle at (250,280)-(271,301): text "IN8"; alarm colour if IN8
rectangle at (300,160)-(321,181): text "IN9"; alarm colour if IN9
rectangle at (290,110)-(361,141): text "Vstupy 2"
rectangle at (330,160)-(351,181): text "IN10"; alarm colour if VzdalenyVstup2
rectangle at (290,130)-(361,161): text "750-430"
rectangle at (300,200)-(321,221): text "IN11"; alarm colour if IN11
rectangle at (330,200)-(351,221): text "IN12"; alarm colour if IN12
rectangle at (300,240)-(321,261): text "IN13"; alarm colour if IN13
rectangle at (330,240)-(351,261): text "IN14"; alarm colour if IN14
rectangle at (300,280)-(321,301): text "IN15"; alarm colour if IN15
rectangle at (330,280)-(351,301): text "IN16"; alarm colour if IN16
rectangle at (220,440)-(241,461): text "IN1"; alarm colour if Host1IN1
rectangle at (210,390)-(281,421): text "Vstupy 1"
rectangle at (250,440)-(271,461): text "IN2"; alarm colour if Host1IN2
rectangle at (210,410)-(281,441): text "750-430"
rectangle at (10,370)-(201,401): text "750-352"
rectangle at (10,390)-(191,421): text "IP adresa vzdálené stanice:"
rectangle at (20,440)-(191,471): text "%s"; shows IPHost1
rectangle at (220,480)-(241,501): text "IN3"; alarm colour if Host1IN3
rectangle at (250,480)-(271,501): text "IN4"; alarm colour if Host1IN4
rectangle at (220,520)-(241,541): text "IN5"; alarm colour if Host1IN5
rectangle at (250,520)-(271,541): text "IN6"; alarm colour if Host1IN6
rectangle at (220,560)-(241,581): text "IN7"; alarm colour if Host1IN7
rectangle at (250,560)-(271,581): text "IN8"; alarm colour if Host1IN8
rectangle at (620,440)-(641,461): text "IN1"; alarm colour if Host2IN1
rectangle at (610,390)-(681,421): text "Vstupy 1"
rectangle at (650,440)-(671,461): text "IN2"; alarm colour if Host2IN2
rectangle at (610,410)-(681,441): text "750-430"
rectangle at (410,370)-(601,401): text "750-352"
rectangle at (410,390)-(591,421): text "IP adresa vzdálené stanice:"
rectangle at (420,440)-(591,471): text "%s"; shows IPHost2
rectangle at (620,480)-(641,501): text "IN3"; alarm colour if Host2IN3
rectangle at (650,480)-(671,501): text "IN4"; alarm colour if Host2IN4
rectangle at (620,520)-(641,541): text "IN5"; alarm colour if Host2IN5
rectangle at (650,520)-(671,541): text "IN6"; alarm colour if Host2IN6
rectangle at (620,560)-(641,581): text "IN7"; alarm colour if Host2IN7
rectangle at (650,560)-(671,581): text "IN8"; alarm colour if Host2IN8
rectangle at (0,40)-(801,81): text "SLEVARNA AL OJS I"
rectangle at (0,320)-(421,361): text "SLEVARNA AL OJS II"
rectangle at (410,320)-(801,361): text "SLEVARNA AL OJS III"
button at (710,0)-(791,31): text "Zpet"; opens plc_vizu
rectangle at (700,440)-(721,461): text "IN9"; alarm colour if Host2IN9
rectangle at (690,390)-(761,421): text "Vstupy 2"
rectangle at (730,440)-(751,461): text "IN10"; alarm colour if Host2IN10
rectangle at (690,410)-(761,441): text "750-430"
rectangle at (700,480)-(721,501): text "IN11"; alarm colour if Host2IN11
rectangle at (730,480)-(751,501): text "IN12"; alarm colour if Host2IN12
rectangle at (700,520)-(721,541): text "IN13"; alarm colour if Host2IN13
rectangle at (730,520)-(751,541): text "IN14"; alarm colour if Host2IN14
rectangle at (700,560)-(721,581): text "IN15"; alarm colour if Host2IN15
rectangle at (730,560)-(751,581): text "IN16"; alarm colour if Host2IN16
19 more shapes without text or variables
*)

(* Visualisation Slitina
